NETWORK
TITLE =R5_Kreislauf_ohne_aussen  Rinser CIP-Kreis ohne pulsierenden
// Act 006
// Box           : Rinser5
// Output address: Q172.3
      CALL FC    70 (
           UnitNo                   := #UnitNo,
           ActRec                   := DB2650.R5_Kreislauf_ohne_aussen,
           Typ                      := 0,
           FBa                      := #xTmp,
           FBa2                     := #xTmp,
           Out                      := Q    172.3);

NETWORK
TITLE =R5_Kreislauf_mit_aussen  Rinser CIP-Kreis mit pulsierenden
// Act 007
// Box           : Rinser5
// Output address: Q172.4
      CALL FC    70 (
           UnitNo                   := #UnitNo,
           ActRec                   := DB2650.R5_Kreislauf_mit_aussen,
           Typ                      := 0,
           FBa                      := #xTmp,
           FBa2                     := #xTmp,
           Out                      := Q    172.4);

NETWORK
TITLE =R5_Grundstellung  Rinser A5 Maschine Grundstellung (Impuls)
// Act 008
// Box           : Rinser5
// Output address: Q172.2
      CALL FC    70 (
           UnitNo                   := #UnitNo,
           ActRec                   := DB2650.R5_Grundstellung,
           Typ                      := 0,
           FBa                      := #xTmp,
           FBa2                     := #xTmp,
           Out                      := Q    172.2);

NETWORK
TITLE =R5_Drainagestellung  Rinser A5 Drainagestellung (Impuls)
// Act 009
// Box           : Rinser5
// Output address: Q172.5
      CALL FC    70 (
           UnitNo                   := #UnitNo,
           ActRec                   := DB2650.R5_Drainagestellung,
           Typ                      := 0,
           FBa                      := #xTmp,
           FBa2                     := #xTmp,
           Out                      := Q    172.5);

NETWORK
TITLE =F5_Kreislauf_o_puls  Füller CIP-Kreis ohne pulsierenden Ablauf
// Act 010
// Box           : Füller5
// Output address: Q196.2
      CALL FC    70 (
           UnitNo                   := #UnitNo,
           ActRec                   := DB2650.F5_Kreislauf_o_puls,
           Typ                      := 0,
           FBa                      := #xTmp,
           FBa2                     := #xTmp,
           Out                      := Q    196.2);

NETWORK
TITLE =F5_Kreislauf_m_puls  Füller CIP-Kreis mit pulsierenden Ablauf
// Act 011
// Box           : Füller5
// Output address: Q196.3
      CALL FC    70 (
           UnitNo                   := #UnitNo,
           ActRec                   := DB2650.F5_Kreislauf_m_puls,
           Typ                      := 0,
           FBa                      := #xTmp,
           FBa2                     := #xTmp,
           Out                      := Q    196.3);

NETWORK
TITLE =F5_Randvollstellung  Füller A5 Randvollstellung Standdesinfektio
// Act 012
// Box           : Füller5
// Output address: Q196.4
      CALL FC    70 (
           UnitNo                   := #UnitNo,
           ActRec                   := DB2650.F5_Randvollstellung,
           Typ                      := 0,
           FBa                      := #xTmp,
           FBa2                     := #xTmp,
           Out                      := Q    196.4);

NETWORK
TITLE =F5_Klarspuelen_o_CIP_Beh  Füller A5 Klarspülen ohne CIP-Behälter
// Act 013
// Box           : Füller5
// Output address: Q196.5
      CALL FC    70 (
           UnitNo                   := #UnitNo,
           ActRec                   := DB2650.F5_Klarspuelen_o_CIP_Beh,
           Typ                      := 0,
           FBa                      := #xTmp,
           FBa2                     := #xTmp,
           Out                      := Q    196.5);

NETWORK
TITLE =F5_Ausschub_m_Sterilluft  Füller Ausschubprogramm mit Sterilluft
// Act 014
// Box           : Füller5
// Output address: Q196.6
      CALL FC    70 (
           UnitNo                   := #UnitNo,
           ActRec                   := DB2650.F5_Ausschub_m_Sterilluft,
           Typ                      := 0,
           FBa                      := #xTmp,
           FBa2                     := #xTmp,
           Out                      := Q    196.6);

NETWORK
TITLE =F5_Ausschub_m_CO2  Füller A5 Ausschubprogramm mit CO2
// Act 015
// Box           : Füller5
// Output address: Q196.7
      CALL FC    70 (
           UnitNo                   := #UnitNo,
           ActRec                   := DB2650.F5_Ausschub_m_CO2,
           Typ                      := 0,
           FBa                      := #xTmp,
           FBa2                     := #xTmp,
           Out                      := Q    196.7);

NETWORK
TITLE =F5_Grundstellung  Füller A5 Maschine Grundstellung (Impuls)
// Act 016
// Box           : Füller5
// Output address: Q197.0
      CALL FC    70 (
           UnitNo                   := #UnitNo,
           ActRec                   := DB2650.F5_Grundstellung,
           Typ                      := 0,
           FBa                      := #xTmp,
           FBa2                     := #xTmp,
           Out                      := Q    197.0);

NETWORK
TITLE =F5_Drainagestellung  Füller A5 Drainagestellung (Impuls)
// Act 017
// Box           : Füller5
// Output address: Q197.1
      CALL FC    70 (
           UnitNo                   := #UnitNo,
           ActRec                   := DB2650.F5_Drainagestellung,
           Typ                      := 0,
           FBa                      := #xTmp,
           FBa2                     := #xTmp,
           Out                      := Q    197.1);

NETWORK
TITLE =F5_Bypass  Füller A5 Bypass (Impuls)
// Act 018
// Box           : Füller5
// Output address: Q197.2
      CALL FC    70 (
           UnitNo                   := #UnitNo,
           ActRec                   := DB2650.F5_Bypass,
           Typ                      := 0,
           FBa                      := #xTmp,
           FBa2                     := #xTmp,
           Out                      := Q    197.2);

NETWORK
TITLE =A5_RR1  Reinigungsrücklauf Anlage 5 zu Kreis 1
// Act 020
// Box           : VSRR1-3
// Input address : I84.0
// Output address: Q84.0
      CALL FC    70 (
           UnitNo                   := #UnitNo,
           ActRec                   := DB2650.A5_RR1,
           Typ                      := 1,
           FBa                      := #xTmp,
           FBa2                     := I     84.0,
           Out                      := Q     84.0);

NETWORK
TITLE =A5_RR2  Reinigungsrücklauf Anlage 5 zu Kreis 2
// Act 021
// Box           : VSRR1-3
// Input address : I84.1
// Output address: Q84.1
      CALL FC    70 (
           UnitNo                   := #UnitNo,
           ActRec                   := DB2650.A5_RR2,
           Typ                      := 1,
           FBa                      := #xTmp,
           FBa2                     := I     84.1,
           Out                      := Q     84.1);

NETWORK
TITLE =A5_RR3  Reinigungsrücklauf Anlage 5 zu Kreis 3
// Act 022
// Box           : VSRR1-3
// Input address : I84.2
// Output address: Q84.2
      CALL FC    70 (
           UnitNo                   := #UnitNo,
           ActRec                   := DB2650.A5_RR3,
           Typ                      := 1,
           FBa                      := #xTmp,
           FBa2                     := I     84.2,
           Out                      := Q     84.2);

NETWORK
TITLE =M5_Grundstellung  Mixer A5 Grundstellung (Impuls)
// Act 023
// Box           : Mixer5
// Output address: Q198.0
      CALL FC    70 (
           UnitNo                   := #UnitNo,
           ActRec                   := DB2650.M5_Grundstellung,
           Typ                      := 0,
           FBa                      := #xTmp,
           FBa2                     := #xTmp,
           Out                      := Q    198.0);

NETWORK
TITLE =M5_Drainagestellung  Mixer A5 Drainagestellung (Impuls)
// Act 024
// Box           : Mixer5
// Output address: Q198.1
      CALL FC    70 (
           UnitNo                   := #UnitNo,
           ActRec                   := DB2650.M5_Drainagestellung,
           Typ                      := 0,
           FBa                      := #xTmp,
           FBa2                     := #xTmp,
           Out                      := Q    198.1);

NETWORK
TITLE =M5_Ausspritzen_o_Ablauf  MixerAusspritzen ohne Ablauf
// Act 025
// Box           : Mixer5
// Output address: Q198.2
      CALL FC    70 (
           UnitNo                   := #UnitNo,
           ActRec                   := DB2650.M5_Ausspritzen_o_Ablauf,
           Typ                      := 0,
           FBa                      := #xTmp,
           FBa2                     := #xTmp,
           Out                      := Q    198.2);

NETWORK
TITLE =M5_Ausspritzen_m_Ablauf  Mixer A5 Ausspritzen mit Ablauf (Impuls
// Act 026
// Box           : Mixer5
// Output address: Q198.3
      CALL FC    70 (
           UnitNo                   := #UnitNo,
           ActRec                   := DB2650.M5_Ausspritzen_m_Ablauf,
           Typ                      := 0,
           FBa                      := #xTmp,
           FBa2                     := #xTmp,
           Out                      := Q    198.3);

NETWORK
TITLE =M5_Fluten_o_Ablauf  Mixer A5 Fluten ohne Ablauf (Impuls)
// Act 027
// Box           : Mixer5
// Output address: Q198.4
      CALL FC    70 (
           UnitNo                   := #UnitNo,
           ActRec                   := DB2650.M5_Fluten_o_Ablauf,
           Typ                      := 0,
           FBa                      := #xTmp,
           FBa2                     := #xTmp,
           Out                      := Q    198.4);

NETWORK
TITLE =M5_Fluten_m_Ablauf  Mixer A5 Fluten mit Ablauf (Impuls)
// Act 028
// Box           : Mixer5
// Output address: Q198.5
      CALL FC    70 (
           UnitNo                   := #UnitNo,
           ActRec                   := DB2650.M5_Fluten_m_Ablauf,
           Typ                      := 0,
           FBa                      := #xTmp,
           FBa2                     := #xTmp,
           Out                      := Q    198.5);

NETWORK
TITLE =M5_Randvollstellung  Mixer A5 Randvollstellung (Impuls)
// Act 029
// Box           : Mixer5
// Output address: Q198.6
      CALL FC    70 (
           UnitNo                   := #UnitNo,
           ActRec                   := DB2650.M5_Randvollstellung,
           Typ                      := 0,
           FBa                      := #xTmp,
           FBa2                     := #xTmp,
           Out                      := Q    198.6);

NETWORK
TITLE =M5_Abpumpen  Mixer A5 Abpumpen (Impuls)
// Act 030
// Box           : Mixer5
// Output address: Q198.7
      CALL FC    70 (
           UnitNo                   := #UnitNo,
           ActRec                   := DB2650.M5_Abpumpen,
           Typ                      := 0,
           FBa                      := #xTmp,
           FBa2                     := #xTmp,
           Out                      := Q    198.7);

NETWORK
TITLE =M5_Klarspuelen  Mixer A5 Klarspülen
// Act 031
// Box           : Mixer5
// Output address: Q199.0
      CALL FC    70 (
           UnitNo                   := #UnitNo,
           ActRec                   := DB2650.M5_Klarspuelen,
           Typ                      := 0,
           FBa                      := #xTmp,
           FBa2                     := #xTmp,
           Out                      := Q    199.0);

END_FUNCTION_BLOCK

FUNCTION_BLOCK FB 1651
TITLE =U065: Packaging Plant 5
FAMILY : BOTEC_F1
NAME : UniE
VERSION : 1.2


VAR_TEMP
  CIP : BOOL ;	//CIP active
  UNIM : BOOL ;	//Unit Not In Maintenance
  GenRel : BOOL ;	//general OK (emergency and maintenance OK)
  EStopOK : BOOL ;	//emergency OK
  UnitNo : INT ;	//unit number
  xTmp : BOOL ;	//Temporary Bool
  iTmp : INT ;	//Temporary INT
  rTmp : REAL ;	//Temporary REAL
  dTmp : DINT ;	//Temporary DINT (free for general use)
  RetValInt : INT ;	//return value
END_VAR
BEGIN
NETWORK
TITLE =General

      SET   ;
// Simulation ---------------------------------------------------------------
      A     DB1651.DBX 1357.7;
      CC    FB  1659; // "U065Sim"
      A     DB1651.DBX   17.3;
      =     DB1651.DBX 1357.7; //Help bit for simulation

// get unit number ----------------------------------------------------------
      L     DB1650.DBW    0;
      T     #UnitNo;

// CIP ----------------------------------------------------------------------
      L     DB1651.DBD   54;
      L     0;
      <D    ;
      =     #CIP;

// emergency OK -------------------------------------------------------------
      A     DB1655.DBX   27.0; //Emergency Stop OK
      =     #EStopOK;

// Write Unit in Maintenance ------------------------------------------------

      AN    DB1651.DBX   69.7;
      =     #UNIM;

// emergency and maintenance OK ---------------------------------------------
      A     #EStopOK;
      A     #UNIM;
      =     #GenRel;

// communication ------------------------------------------------------------
      UC    FB  1655; // U065Com

NETWORK
TITLE =Analog Inputs

      NOP   0;

// ----------------------------------------------------------
// A5_TI1
// ----------------------------------------------------------
//      L     ID   352
//      T     "U065AnID".A5_TI1.ValRaw
      SET   ;
      R     DB2653.DBX  143.5;

      L     DB1651.DBD 1118; // !!! insert correct SFM !!!
      T     DB2653.DBD  238;

      SET   ;
      =     DB2653.DBX  141.5;


NETWORK
TITLE =Universal Value

      NOP   0;

// ----------------------------------------------------------
// unv001 Process Status
// ----------------------------------------------------------
// process value to UnV
//      L     0.000000e+000
//      T     "U065UnVD".unv001.ValExt

// ----------------------------------------------------------
// unv002 Universal Value 02
// ----------------------------------------------------------
// process value to UnV
//      L     0.000000e+000
//      T     "U065UnVD".unv002.ValExt

// ----------------------------------------------------------
// unv003 Universal Value 03
// ----------------------------------------------------------
// process value to UnV
//      L     0.000000e+000
//      T     "U065UnVD".unv003.ValExt

// ----------------------------------------------------------
// unv004 Universal Value 04
// ----------------------------------------------------------
// process value to UnV
//      L     0.000000e+000
//      T     "U065UnVD".unv004.ValExt

NETWORK
TITLE =Special Input

      NOP   0;

// ----------------------------------------------------------
// A5_MIXER_CIP_BEREIT Koppelsignal von Mixer 5 CIP-Bereitschaft (Dauersignal)
// ----------------------------------------------------------
      A     DB2650.DBX  102.6;
      =     DB2651.DBX   81.4;
      SET   ;
      =     DB2651.DBX   81.5;


// ----------------------------------------------------------
// A5_MIXER_VOLL Koppelsignal von Mixer 5 Mixer voll
// ----------------------------------------------------------
//      CLR
//      =     "U065SpID".A5_MIXER_VOLL.EAl
//      =     "U065SpID".A5_MIXER_VOLL.Pre

// ----------------------------------------------------------
// A5_MIXER_LEER Koppelsignal von Mixer 5 Mixer leer
// ----------------------------------------------------------
//      CLR
//      =     "U065SpID".A5_MIXER_LEER.EAl
//      =     "U065SpID".A5_MIXER_LEER.Pre

// ----------------------------------------------------------
// A5_MIXER_Anforderung Koppelsignal von Mixer 5 Anforderung Nachsp.
// ----------------------------------------------------------
//      CLR
//      =     "U065SpID".A5_MIXER_Anforderung.EAl
//      =     "U065SpID".A5_MIXER_Anforderung.Pre

// ----------------------------------------------------------
// M5_WATCHDOG Koppelsignal von Mixer 5 WATCHDOG
// ----------------------------------------------------------
//      CLR
//      =     "U065SpID".M5_WATCHDOG.EAl
//      =     "U065SpID".M5_WATCHDOG.Pre

// ----------------------------------------------------------
// A5_SS_FRG_MOLCH Anlage 5 Schlüsselschalter Freigabe Molch
// ----------------------------------------------------------
//      CLR
//      =     "U065SpID".A5_SS_FRG_MOLCH.EAl
//      =     "U065SpID".A5_SS_FRG_MOLCH.Pre

// ----------------------------------------------------------
// E195_7 Anlage 5 Reserve 7 Ende Ventilschrank A5
// ----------------------------------------------------------
//      CLR
//      =     "U065SpID".E195_7.EAl
//      =     "U065SpID".E195_7.Pre

// ----------------------------------------------------------
// A5_LDT_PROD
// ----------------------------------------------------------
//      CLR
//      =     "U065SpID".A5_LDT_PROD.EAl
//      =     "U065SpID".A5_LDT_PROD.Pre

// ----------------------------------------------------------
// A5_LDT_QUITT_CIP
// ----------------------------------------------------------
//      CLR
//      =     "U065SpID".A5_LDT_QUITT_CIP.EAl
//      =     "U065SpID".A5_LDT_QUITT_CIP.Pre

// ----------------------------------------------------------
// A5_DT_START
// ----------------------------------------------------------
//      CLR
//      =     "U065SpID".A5_DT_START.EAl
//      =     "U065SpID".A5_DT_START.Pre

// ----------------------------------------------------------
// A5_FUELLER_LAEUFT Koppelsignal von Füller 5 Füller läuft (Dauersignal)
// ----------------------------------------------------------
//      CLR
//      =     "U065SpID".A5_FUELLER_LAEUFT.EAl
//      =     "U065SpID".A5_FUELLER_LAEUFT.Pre

// ----------------------------------------------------------
// A5_FUELLER_LEER Koppelsignal von Füller 5 Füller leer (Impuls)
// ----------------------------------------------------------
//      CLR
//      =     "U065SpID".A5_FUELLER_LEER.EAl
//      =     "U065SpID".A5_FUELLER_LEER.Pre

// ----------------------------------------------------------
// A5_FUELLER_VOLL Koppelsignal von Füller 5 Füller voll (Impuls)
// ----------------------------------------------------------
//      CLR
//      =     "U065SpID".A5_FUELLER_VOLL.EAl
//      =     "U065SpID".A5_FUELLER_VOLL.Pre

// ----------------------------------------------------------
// A5_FUELLER_KLARSPUELEN Koppelsignal von Füller 5 Klarspülen
// ----------------------------------------------------------
//      CLR
//      =     "U065SpID".A5_FUELLER_KLARSPUELEN.EAl
//      =     "U065SpID".A5_FUELLER_KLARSPUELEN.Pre

// ----------------------------------------------------------
// F5_WATCHDOG Koppelsignal von Füller 5 WATCHDOG
// ----------------------------------------------------------
//      CLR
//     =     "U065SpID".F5_WATCHDOG.EAl
//     =     "U065SpID".F5_WATCHDOG.Pre

// ----------------------------------------------------------
// A5_RINSER_LAEUFT Koppelsignal von Rinser 5 Rinser läuft (Dauersignal)
// ----------------------------------------------------------
//      CLR
//      =     "U065SpID".A5_RINSER_LAEUFT.EAl
//      =     "U065SpID".A5_RINSER_LAEUFT.Pre

// ----------------------------------------------------------
// R5_WATCHDOG Koppelsignal von Rinser 5 WATCHDOG
// ----------------------------------------------------------
//      CLR
//      =     "U065SpID".R5_WATCHDOG.EAl
//      =     "U065SpID".R5_WATCHDOG.Pre

NETWORK
TITLE =Messages

      NOP   0;

// ----------------------------------------------------------
// msg001 Message 01
// ----------------------------------------------------------
      SET   ;
      R     DB2657.DBX   80.7;
      =     DB2657.DBX   81.4;

      CLR   ;
      =     DB2657.DBX   82.7;

// ----------------------------------------------------------
// msg002 Message 02
// ----------------------------------------------------------
      SET   ;
      R     DB2657.DBX  140.7;
      =     DB2657.DBX  141.4;

      CLR   ;
      =     DB2657.DBX  142.7;

// ----------------------------------------------------------
// msg003 Message 03
// ----------------------------------------------------------
      SET   ;
      R     DB2657.DBX  200.7;
      =     DB2657.DBX  201.4;

      CLR   ;
      =     DB2657.DBX  202.7;

NETWORK
TITLE =Sequence organisation

      CLR   ;
      =     M    122.2;

// SFM supply ----------------------------------------------------------------

// analog value to SFM spare -----------------------
      L     DB2653.DBD  146;
      T     DB1651.DBD 1122; // !!! insert correct SFM !!!

// sequencer ----------------------------------------------------------------
      A     DB1653.DBX   43.1;
      S     DB1653.DBX   97.3;

      CALL FC    40 (
           UnitNo                   := #UnitNo);

NETWORK
TITLE =Auto / Manual

      SET   ;
      AN    M    122.2;
      JC    MODE;
      AN    M    120.1;

// assign actuator mode
      AN    M    120.1;
      =     DB2650.DBX  105.4;
      =     DB2650.DBX  185.4;
      S     DB2650.DBX  265.4;
      =     DB2650.DBX  345.4;
      S     DB2650.DBX  425.4;
      =     DB2650.DBX  505.4;
      =     DB2650.DBX  585.4;
      =     DB2650.DBX  665.4;
      =     DB2650.DBX  745.4;
      =     DB2650.DBX  825.4;
      =     DB2650.DBX  905.4;
      =     DB2650.DBX  985.4;
      =     DB2650.DBX 1065.4;
      =     DB2650.DBX 1145.4;
      =     DB2650.DBX 1225.4;
      =     DB2650.DBX 1305.4;
      =     DB2650.DBX 1385.4;
      =     DB2650.DBX 1465.4;
      =     DB2650.DBX 1545.4;
      =     DB2650.DBX 1625.4;
      =     DB2650.DBX 1705.4;
      =     DB2650.DBX 1785.4;
      =     DB2650.DBX 1865.4;
      =     DB2650.DBX 1945.4;
      =     DB2650.DBX 2025.4;
      =     DB2650.DBX 2105.4;
      =     DB2650.DBX 2185.4;
      =     DB2650.DBX 2265.4;
      =     DB2650.DBX 2345.4;
      =     DB2650.DBX 2425.4;
      =     DB2650.DBX 2505.4;




MODE: SET   ;

NETWORK
TITLE =A5_RP1 Rücklaufpumpe Anlage 5
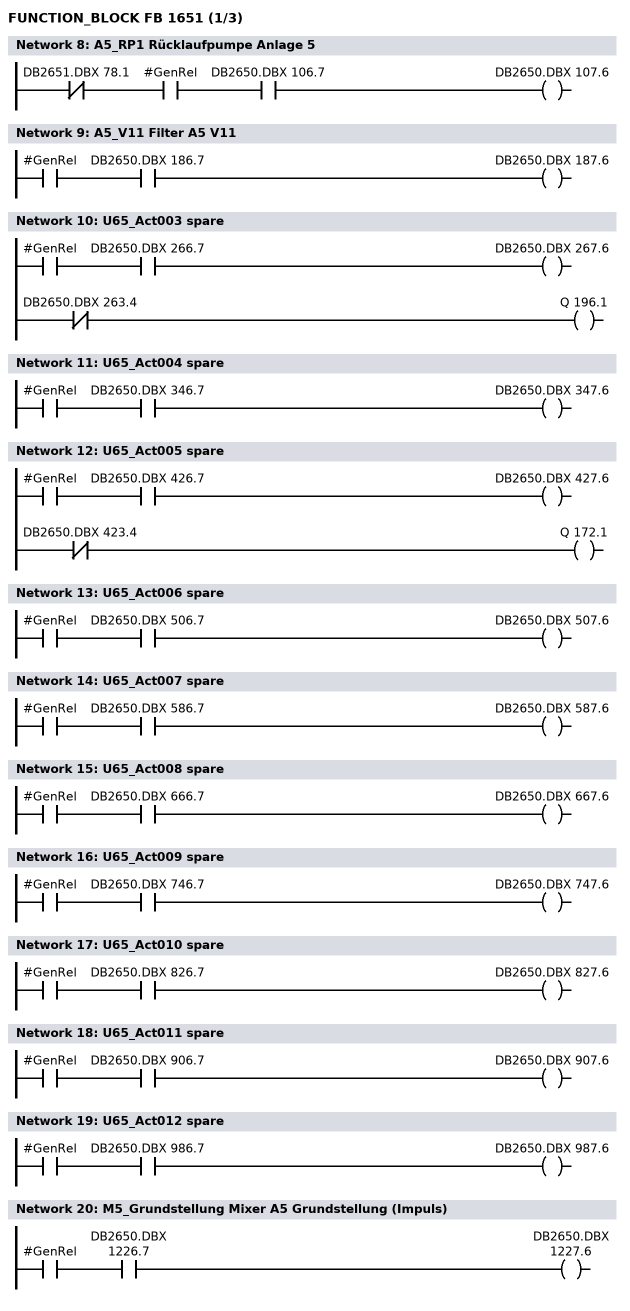

//      A     "U065SpID".A5_FS1.Sig
      AN    DB2651.DBX   78.1;

      A     #GenRel;
      A     DB2650.DBX  106.7;
      =     DB2650.DBX  107.6;
NETWORK
TITLE =A5_V11 Filter A5 V11

      A     #GenRel;
      A     DB2650.DBX  186.7;
      =     DB2650.DBX  187.6;
NETWORK
TITLE =U65_Act003 spare

      A     #GenRel;
      A     DB2650.DBX  266.7;
      =     DB2650.DBX  267.6;

      AN    DB2650.DBX  263.4;
      =     Q    196.1;
NETWORK
TITLE =U65_Act004 spare

      A     #GenRel;
      A     DB2650.DBX  346.7;
      =     DB2650.DBX  347.6;
NETWORK
TITLE =U65_Act005 spare

      A     #GenRel;
      A     DB2650.DBX  426.7;
      =     DB2650.DBX  427.6;

      AN    DB2650.DBX  423.4;
      =     Q    172.1;
NETWORK
TITLE =U65_Act006 spare

      A     #GenRel;
      A     DB2650.DBX  506.7;
      =     DB2650.DBX  507.6;
NETWORK
TITLE =U65_Act007 spare

      A     #GenRel;
      A     DB2650.DBX  586.7;
      =     DB2650.DBX  587.6;
NETWORK
TITLE =U65_Act008 spare

      A     #GenRel;
      A     DB2650.DBX  666.7;
      =     DB2650.DBX  667.6;
NETWORK
TITLE =U65_Act009 spare

      A     #GenRel;
      A     DB2650.DBX  746.7;
      =     DB2650.DBX  747.6;
NETWORK
TITLE =U65_Act010 spare

      A     #GenRel;
      A     DB2650.DBX  826.7;
      =     DB2650.DBX  827.6;
NETWORK
TITLE =U65_Act011 spare

      A     #GenRel;
      A     DB2650.DBX  906.7;
      =     DB2650.DBX  907.6;
NETWORK
TITLE =U65_Act012 spare

      A     #GenRel;
      A     DB2650.DBX  986.7;
      =     DB2650.DBX  987.6;
NETWORK
TITLE =M5_Grundstellung Mixer A5 Grundstellung (Impuls)

      A     #GenRel;
      A     DB2650.DBX 1226.7;
      =     DB2650.DBX 1227.6;
NETWORK
TITLE =M5_Drainagestellung Mixer A5 Drainagestellung (Impuls)
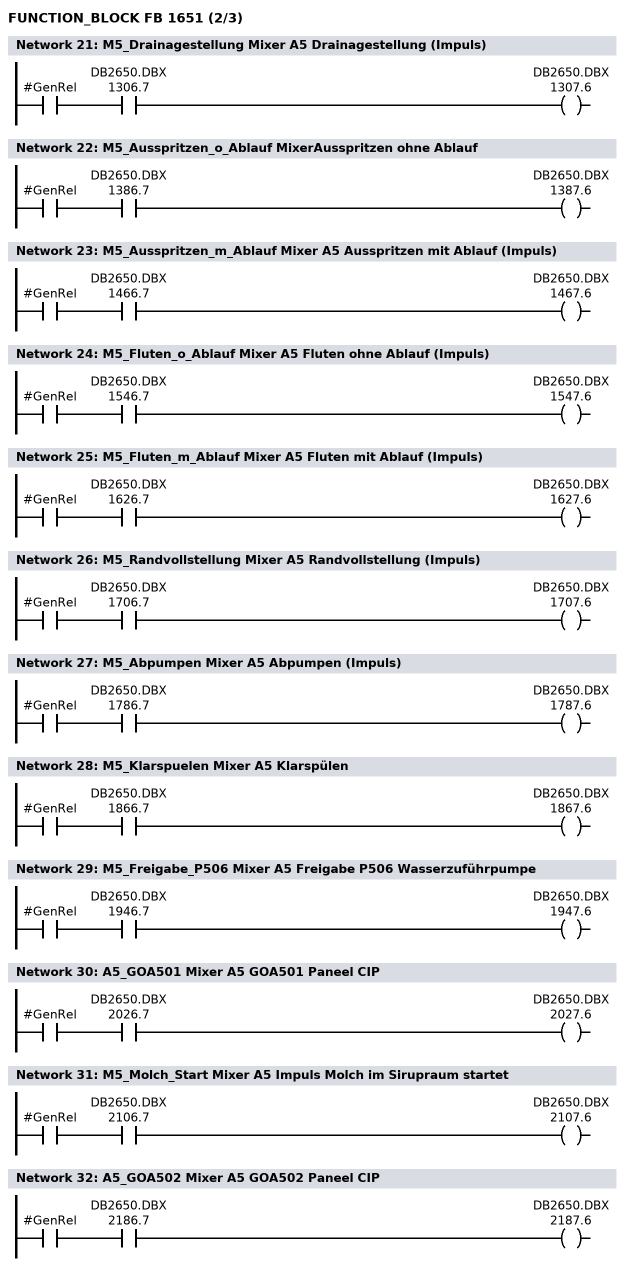

      A     #GenRel;
      A     DB2650.DBX 1306.7;
      =     DB2650.DBX 1307.6;
NETWORK
TITLE =M5_Ausspritzen_o_Ablauf MixerAusspritzen ohne Ablauf

      A     #GenRel;
      A     DB2650.DBX 1386.7;
      =     DB2650.DBX 1387.6;
NETWORK
TITLE =M5_Ausspritzen_m_Ablauf Mixer A5 Ausspritzen mit Ablauf (Impuls)

      A     #GenRel;
      A     DB2650.DBX 1466.7;
      =     DB2650.DBX 1467.6;
NETWORK
TITLE =M5_Fluten_o_Ablauf Mixer A5 Fluten ohne Ablauf (Impuls)

      A     #GenRel;
      A     DB2650.DBX 1546.7;
      =     DB2650.DBX 1547.6;
NETWORK
TITLE =M5_Fluten_m_Ablauf Mixer A5 Fluten mit Ablauf (Impuls)

      A     #GenRel;
      A     DB2650.DBX 1626.7;
      =     DB2650.DBX 1627.6;
NETWORK
TITLE =M5_Randvollstellung Mixer A5 Randvollstellung (Impuls)

      A     #GenRel;
      A     DB2650.DBX 1706.7;
      =     DB2650.DBX 1707.6;
NETWORK
TITLE =M5_Abpumpen Mixer A5 Abpumpen (Impuls)

      A     #GenRel;
      A     DB2650.DBX 1786.7;
      =     DB2650.DBX 1787.6;
NETWORK
TITLE =M5_Klarspuelen Mixer A5 Klarspülen

      A     #GenRel;
      A     DB2650.DBX 1866.7;
      =     DB2650.DBX 1867.6;
NETWORK
TITLE =M5_Freigabe_P506 Mixer A5 Freigabe P506 Wasserzuführpumpe

      A     #GenRel;
      A     DB2650.DBX 1946.7;
      =     DB2650.DBX 1947.6;
NETWORK
TITLE =A5_GOA501 Mixer A5 GOA501 Paneel CIP

      A     #GenRel;
      A     DB2650.DBX 2026.7;
      =     DB2650.DBX 2027.6;
NETWORK
TITLE =M5_Molch_Start Mixer A5 Impuls Molch im Sirupraum startet

      A     #GenRel;
      A     DB2650.DBX 2106.7;
      =     DB2650.DBX 2107.6;
NETWORK
TITLE =A5_GOA502 Mixer A5 GOA502 Paneel CIP

      A     #GenRel;
      A     DB2650.DBX 2186.7;
      =     DB2650.DBX 2187.6;
NETWORK
TITLE =A5_GOA503 Mixer A5 GOA503 Paneel CIP
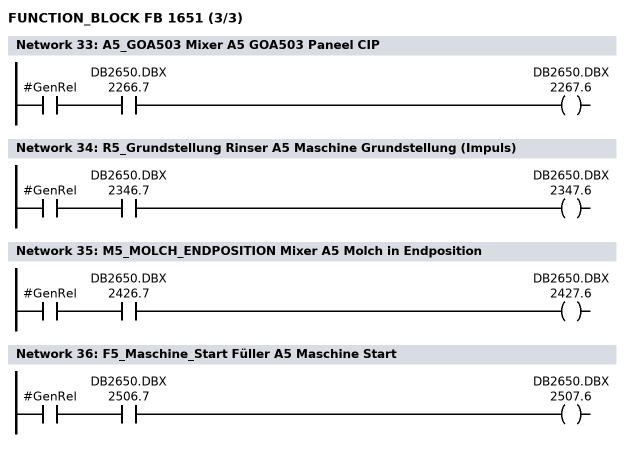

      A     #GenRel;
      A     DB2650.DBX 2266.7;
      =     DB2650.DBX 2267.6;
NETWORK
TITLE =R5_Grundstellung Rinser A5 Maschine Grundstellung (Impuls)

      A     #GenRel;
      A     DB2650.DBX 2346.7;
      =     DB2650.DBX 2347.6;
NETWORK
TITLE =M5_MOLCH_ENDPOSITION Mixer A5 Molch in Endposition

      A     #GenRel;
      A     DB2650.DBX 2426.7;
      =     DB2650.DBX 2427.6;
NETWORK
TITLE =F5_Maschine_Start Füller A5 Maschine Start

      A     #GenRel;
      A     DB2650.DBX 2506.7;
      =     DB2650.DBX 2507.6;
END_FUNCTION_BLOCK

FUNCTION_BLOCK FB 1670
TITLE =U067: Abfüllanlage  7
FAMILY : BOTEC_F1
NAME : U067A
VERSION : 2.1


VAR_TEMP
  EStopOK : BOOL ;	//auxiliary flag
  CIP : BOOL ;	//CIP Program Selected
  xTmp : BOOL ;	//Temporary Bool(free for general use)
  DummyBool : BOOL ;	//Temporary Bool(free for general use)
  UnitNo : INT ;	//unit number
  UnitFB : INT ;	//unit expansion FB number
  rTmp : REAL ;	//Temporary REAL (free for general use)
  iTmp : INT ;	//Temporary INT (free for general use)
  DummyInt : INT ;	//Temporary INT (free for general use)
  dTmp : DINT ;	//Temporary DINT (free for general use)
END_VAR
BEGIN
NETWORK
TITLE =general

      CLR   ;
      =     #xTmp;
      =     #EStopOK;

      L     DB1670.DBW    0;
      T     #UnitNo;
      L     DB1670.DBW    2;
      T     #UnitFB;

NETWORK
TITLE =Universal value

      NOP   0;
// unv001 UnV 001 Process Status
      CALL FC    27 (
           UnitNo                   := #UnitNo,
           UnVRec                   := DB2675.unv001,
           ValExt                   := DB2675.DBD  234);

// unv002 UnV 002 Universal Value 02
      CALL FC    27 (
           UnitNo                   := #UnitNo,
           UnVRec                   := DB2675.unv002,
           ValExt                   := DB2675.DBD  362);

// unv003 UnV 003 Universal Value 03
      CALL FC    27 (
           UnitNo                   := #UnitNo,
           UnVRec                   := DB2675.unv003,
           ValExt                   := DB2675.DBD  490);

// unv004 UnV 004 Universal Value 04
      CALL FC    27 (
           UnitNo                   := #UnitNo,
           UnVRec                   := DB2675.unv004,
           ValExt                   := DB2675.DBD  618);

NETWORK
TITLE =special inputs

      NOP   0;
// FS_A7FS1 SpI 001 STROEMUNGSSCHALTER A7
      CALL FC    14 (
           UnitNo                   := #UnitNo,
           SpIRec                   := DB2671.FS_A7FS1,
           SpIBit                   := I     27.0);

// A7_FUELLER_LAEUFT SpI 002 Fueller 7 laeuft
      CALL FC    14 (
           UnitNo                   := #UnitNo,
           SpIRec                   := DB2671.A7_FUELLER_LAEUFT,
           SpIBit                   := I     76.1);

// A7_MIXER_CIP_BEREIT SpI 003 Mixer Anlage 7 CIP-Bereit
      CALL FC    14 (
           UnitNo                   := #UnitNo,
           SpIRec                   := DB2671.A7_MIXER_CIP_BEREIT,
           SpIBit                   := I     78.0);

// A7_MIXER_VOLL SpI 004 Mixer Anlage 7 voll
      CALL FC    14 (
           UnitNo                   := #UnitNo,
           SpIRec                   := DB2671.A7_MIXER_VOLL,
           SpIBit                   := I     78.2);

// A7_MIXER_LEER SpI 005 Mixer Anlage 7 leer
      CALL FC    14 (
           UnitNo                   := #UnitNo,
           SpIRec                   := DB2671.A7_MIXER_LEER,
           SpIBit                   := I     78.1);

// A7_MIXER_ANF_SIRUP SpI 006 Mixer Anlage 7 Anforderung Sirup
      CALL FC    14 (
           UnitNo                   := #UnitNo,
           SpIRec                   := DB2671.A7_MIXER_ANF_SIRUP,
           SpIBit                   := I     78.3);

// A7_FUELLER_CIP_BEREIT SpI 007 Fueller 7 CIP-Bereit
      CALL FC    14 (
           UnitNo                   := #UnitNo,
           SpIRec                   := DB2671.A7_FUELLER_CIP_BEREIT,
           SpIBit                   := I     76.0);

// A7_SS_FRG_MOLCH SpI 009 Anlage 7 Schlüsselschalter Freigabe Molch
      CALL FC    14 (
           UnitNo                   := #UnitNo,
           SpIRec                   := DB2671.A7_SS_FRG_MOLCH,
           SpIBit                   := I     27.4);

// A7_FUELLER_LEER SpI 011 Fueller 7 leer (Impuls)
      CALL FC    14 (
           UnitNo                   := #UnitNo,
           SpIRec                   := DB2671.A7_FUELLER_LEER,
           SpIBit                   := I     76.2);

// GOA_703 SpI 012 Meldung an Fueller/Mixer Anl.7
      CALL FC    14 (
           UnitNo                   := #UnitNo,
           SpIRec                   := DB2671.A7_FUELLER_VOLL,
           SpIBit                   := I     76.3);//"GOA_703"

// A7_RINSER_CIP_BEREIT SpI 013 Rinser Anlage 7 CIP-Bereit
      CALL FC    14 (
           UnitNo                   := #UnitNo,
           SpIRec                   := DB2671.A7_RINSER_CIP_BEREIT,
           SpIBit                   := I     77.0);

// A7_RINSER_LAEUFT SpI 014 Rinser Anlage 7 laeuft
      CALL FC    14 (
           UnitNo                   := #UnitNo,
           SpIRec                   := DB2671.A7_RINSER_LAEUFT,
           SpIBit                   := I     77.1);

// EA7_K1_Handklappe SpI 015 Handklappe Fueller 7
      CALL FC    14 (
           UnitNo                   := #UnitNo,
           SpIRec                   := DB2671.EA7_K1_Handklappe,
           SpIBit                   := I     27.1);

NETWORK
TITLE =messages

      NOP   0;
// msg001 Msg 001 Message 01
      CALL FC    16 (
           UnitNo                   := #UnitNo,
           MsgRec                   := DB2677.msg001,
           MsgBit                   := DB2677.DBX   82.7);

// msg002 Msg 002 Message 02
      CALL FC    16 (
           UnitNo                   := #UnitNo,
           MsgRec                   := DB2677.msg002,
           MsgBit                   := DB2677.DBX  142.7);

// msg003 Msg 003 Message 03
      CALL FC    16 (
           UnitNo                   := #UnitNo,
           MsgRec                   := DB2677.msg003,
           MsgBit                   := DB2677.DBX  202.7);

NETWORK
TITLE =unit supply

      UC    FB [#UnitFB];

NETWORK
TITLE =A7_RRP1  CIP Rücklaufpumpe Anlage 7
// Act 001
// Box           : VSA7
// Input address : I25.7
// Output address: Q47.7
      CALL FC    70 (
           UnitNo                   := #UnitNo,
           ActRec                   := DB2670.A7_RRP1,
           Typ                      := 1,
           FBa                      := #xTmp,
           FBa2                     := I     25.7,
           Out                      := Q     47.7);

NETWORK
TITLE =F7_Maschine_Start  Fueller 7 Start
// Act 002
// Box           : FRM-A7
// Output address: Q54.0
      CALL FC    70 (
           UnitNo                   := #UnitNo,
           ActRec                   := DB2670.F7_Maschine_Start,
           Typ                      := 0,
           FBa                      := #xTmp,
           FBa2                     := #xTmp,
           Out                      := Q     54.0);

NETWORK
TITLE =F7_Maschine_Stop  Fueller 7 Stop
// Act 003
// Box           : FRM-A7
// Output address: Q54.1
      CALL FC    70 (
           UnitNo                   := #UnitNo,
           ActRec                   := DB2670.F7_Maschine_Stop,
           Typ                      := 0,
           FBa                      := #xTmp,
           FBa2                     := #xTmp,
           Out                      := #xTmp);

NETWORK
TITLE =R7_START_IMPULS  Rinser 7 Start
// Act 004
// Box           : FRM-A7
// Output address: Q56.0
      CALL FC    70 (
           UnitNo                   := #UnitNo,
           ActRec                   := DB2670.R7_START_IMPULS,
           Typ                      := 0,
           FBa                      := #xTmp,
           FBa2                     := #xTmp,
           Out                      := Q     56.0);

NETWORK
TITLE =R7_STOP  Rinser 7 Stop
// Act 005
// Box           : FRM-A7
// Output address: Q56.1
      CALL FC    70 (
           UnitNo                   := #UnitNo,
           ActRec                   := DB2670.R7_STOP,
           Typ                      := 0,
           FBa                      := #xTmp,
           FBa2                     := #xTmp,
           Out                      := #xTmp);

NETWORK
TITLE =R7_Kreislauf_ohne_aussen  Prog.schritt 15 CIP Krsl.o.ausse.
// Act 006
// Box           : FRM-A7
// Output address: Q56.3
      CALL FC    70 (
           UnitNo                   := #UnitNo,
           ActRec                   := DB2670.R7_Kreislauf_ohne_aussen,
           Typ                      := 0,
           FBa                      := #xTmp,
           FBa2                     := #xTmp,
           Out                      := Q     56.3);

NETWORK
TITLE =R7_Kreislauf_mit_aussen  Prog.schritt 16 CIP Krsl.m.ausse.
// Act 007
// Box           : FRM-A7
// Output address: Q56.4
      CALL FC    70 (
           UnitNo                   := #UnitNo,
           ActRec                   := DB2670.R7_Kreislauf_mit_aussen,
           Typ                      := 0,
           FBa                      := #xTmp,
           FBa2                     := #xTmp,
           Out                      := Q     56.4);

NETWORK
TITLE =R7_Grundstellung  Prog.schritt 1 Grundstellung
// Act 008
// Box           : FRM-A7
// Output address: Q56.2
      CALL FC    70 (
           UnitNo                   := #UnitNo,
           ActRec                   := DB2670.R7_Grundstellung,
           Typ                      := 0,
           FBa                      := #xTmp,
           FBa2                     := #xTmp,
           Out                      := Q     56.2);

NETWORK
TITLE =R7_Drainagestellung  Prog.schritt 2 Drainagestellung
// Act 009
// Box           : FRM-A7
// Output address: Q56.5
      CALL FC    70 (
           UnitNo                   := #UnitNo,
           ActRec                   := DB2670.R7_Drainagestellung,
           Typ                      := 0,
           FBa                      := #xTmp,
           FBa2                     := #xTmp,
           Out                      := Q     56.5);

NETWORK
TITLE =F7_Kreislauf_o_puls  Prog.schritt 15 CIP Krsl.o.ausse.
// Act 010
// Box           : FRM-A7
// Output address: Q54.2
      CALL FC    70 (
           UnitNo                   := #UnitNo,
           ActRec                   := DB2670.F7_Kreislauf_o_puls,
           Typ                      := 0,
           FBa                      := #xTmp,
           FBa2                     := #xTmp,
           Out                      := Q     54.2);

NETWORK
TITLE =F7_Kreislauf_m_puls  Prog.schritt 16 CIP Krsl.m.ausse.
// Act 011
// Box           : FRM-A7
// Output address: Q54.3
      CALL FC    70 (
           UnitNo                   := #UnitNo,
           ActRec                   := DB2670.F7_Kreislauf_m_puls,
           Typ                      := 0,
           FBa                      := #xTmp,
           FBa2                     := #xTmp,
           Out                      := Q     54.3);

NETWORK
TITLE =F7_Randvollstellung  Prog.schritt 17 Randv./Standdes.
// Act 012
// Box           : FRM-A7
// Output address: Q54.4
      CALL FC    70 (
           UnitNo                   := #UnitNo,
           ActRec                   := DB2670.F7_Randvollstellung,
           Typ                      := 0,
           FBa                      := #xTmp,
           FBa2                     := #xTmp,
           Out                      := Q     54.4);

NETWORK
TITLE =F7_Klarspuelen_o_CIP_Beh  Prog.schritt 19 Klarsp.o.CIP Beh
// Act 013
// Box           : FRM-A7
// Output address: Q54.5
      CALL FC    70 (
           UnitNo                   := #UnitNo,
           ActRec                   := DB2670.F7_Klarspuelen_o_CIP_Beh,
           Typ                      := 0,
           FBa                      := #xTmp,
           FBa2                     := #xTmp,
           Out                      := Q     54.5);

NETWORK
TITLE =F7_Ausschub_m_Sterilluft  Prog.schritt 20 Ausschub m.Steri
// Act 014
// Box           : FRM-A7
// Output address: Q54.6
      CALL FC    70 (
           UnitNo                   := #UnitNo,
           ActRec                   := DB2670.F7_Ausschub_m_Sterilluft,
           Typ                      := 0,
           FBa                      := #xTmp,
           FBa2                     := #xTmp,
           Out                      := Q     54.6);

NETWORK
TITLE =F7_Ausschub_m_CO2  Prog.schritt 21 Ausschub m.CO2
// Act 015
// Box           : FRM-A7
// Output address: Q54.7
      CALL FC    70 (
           UnitNo                   := #UnitNo,
           ActRec                   := DB2670.F7_Ausschub_m_CO2,
           Typ                      := 0,
           FBa                      := #xTmp,
           FBa2                     := #xTmp,
           Out                      := Q     54.7);

NETWORK
TITLE =F7_Grundstellung  Prog.schritt 1 Grundstellung
// Act 016
// Box           : FRM-A7
// Output address: Q55.0
      CALL FC    70 (
           UnitNo                   := #UnitNo,
           ActRec                   := DB2670.F7_Grundstellung,
           Typ                      := 0,
           FBa                      := #xTmp,
           FBa2                     := #xTmp,
           Out                      := Q     55.0);

NETWORK
TITLE =F7_Drainagestellung  Prog.schritt 2 Drainagestellung
// Act 017
// Box           : FRM-A7
// Output address: Q55.1
      CALL FC    70 (
           UnitNo                   := #UnitNo,
           ActRec                   := DB2670.F7_Drainagestellung,
           Typ                      := 0,
           FBa                      := #xTmp,
           FBa2                     := #xTmp,
           Out                      := Q     55.1);

NETWORK
TITLE =F7_Bypass  Prog.schritt 30 Bypass
// Act 018
// Box           : FRM-A7
// Output address: Q55.2
      CALL FC    70 (
           UnitNo                   := #UnitNo,
           ActRec                   := DB2670.F7_Bypass,
           Typ                      := 0,
           FBa                      := #xTmp,
           FBa2                     := #xTmp,
           Out                      := Q     55.2);

NETWORK
TITLE =A7_RR1  A7RR1 Ventil CIP Rücklauf Kreis 1 Anlage 7
// Act 020
// Box           : VSRR6-11
// Input address : I28.0
// Output address: Q28.0
      CALL FC    70 (
           UnitNo                   := #UnitNo,
           ActRec                   := DB2670.A7_RR1,
           Typ                      := 1,
           FBa                      := #xTmp,
           FBa2                     := I     28.0,
           Out                      := Q     28.0);

NETWORK
TITLE =A7_RR2  A7RR2 Ventil CIP Rücklauf Kreis 2 Anlage 7
// Act 021
// Box           : VSRR6-11
// Input address : I28.1
// Output address: Q28.1
      CALL FC    70 (
           UnitNo                   := #UnitNo,
           ActRec                   := DB2670.A7_RR2,
           Typ                      := 1,
           FBa                      := #xTmp,
           FBa2                     := I     28.1,
           Out                      := Q     28.1);

NETWORK
TITLE =A7_RR3  A7RR3 Ventil CIP Rücklauf Kreis 3 Anlage 7
// Act 022
// Box           : VSRR6-11
// Input address : I28.2
// Output address: Q28.2
      CALL FC    70 (
           UnitNo                   := #UnitNo,
           ActRec                   := DB2670.A7_RR3,
           Typ                      := 1,
           FBa                      := #xTmp,
           FBa2                     := I     28.2,
           Out                      := Q     28.2);

NETWORK
TITLE =M7_Grundstellung  Prog.schritt 101 Grundstellung
// Act 023
// Box           : FRM-A7
// Output address: Q58.0
      CALL FC    70 (
           UnitNo                   := #UnitNo,
           ActRec                   := DB2670.M7_Grundstellung,
           Typ                      := 0,
           FBa                      := #xTmp,
           FBa2                     := #xTmp,
           Out                      := Q     58.0);

NETWORK
TITLE =M7_Drainagestellung  Prog.schritt 102 Darinage
// Act 024
// Box           : FRM-A7
// Output address: Q58.1
      CALL FC    70 (
           UnitNo                   := #UnitNo,
           ActRec                   := DB2670.M7_Drainagestellung,
           Typ                      := 0,
           FBa                      := #xTmp,
           FBa2                     := #xTmp,
           Out                      := Q     58.1);

NETWORK
TITLE =M7_Ausspritzen_o_Ablauf  Prog.schritt 113 Ausspr.o.Ablauf
// Act 025
// Box           : FRM-A7
// Output address: Q58.2
      CALL FC    70 (
           UnitNo                   := #UnitNo,
           ActRec                   := DB2670.M7_Ausspritzen_o_Ablauf,
           Typ                      := 0,
           FBa                      := #xTmp,
           FBa2                     := #xTmp,
           Out                      := Q     58.2);

NETWORK
TITLE =M7_Ausspritzen_m_Ablauf  Prog.schritt 114 Ausspr.m.Ablauf
// Act 026
// Box           : FRM-A7
// Output address: Q58.3
      CALL FC    70 (
           UnitNo                   := #UnitNo,
           ActRec                   := DB2670.M7_Ausspritzen_m_Ablauf,
           Typ                      := 0,
           FBa                      := #xTmp,
           FBa2                     := #xTmp,
           Out                      := Q     58.3);

NETWORK
TITLE =M7_Fluten_o_Ablauf  Prog.schritt 115 Fluten o.Ablauf
// Act 027
// Box           : FRM-A7
// Output address: Q58.4
      CALL FC    70 (
           UnitNo                   := #UnitNo,
           ActRec                   := DB2670.M7_Fluten_o_Ablauf,
           Typ                      := 0,
           FBa                      := #xTmp,
           FBa2                     := #xTmp,
           Out                      := Q     58.4);

NETWORK
TITLE =M7_Fluten_m_Ablauf  Prog.schritt 116 Fluten m.Ablauf
// Act 028
// Box           : FRM-A7
// Output address: Q58.5
      CALL FC    70 (
           UnitNo                   := #UnitNo,
           ActRec                   := DB2670.M7_Fluten_m_Ablauf,
           Typ                      := 0,
           FBa                      := #xTmp,
           FBa2                     := #xTmp,
           Out                      := Q     58.5);

NETWORK
TITLE =M7_Randvollstellung  Prog.schritt 117 Randvollstellung
// Act 029
// Box           : FRM-A7
// Output address: Q58.6
      CALL FC    70 (
           UnitNo                   := #UnitNo,
           ActRec                   := DB2670.M7_Randvollstellung,
           Typ                      := 0,
           FBa                      := #xTmp,
           FBa2                     := #xTmp,
           Out                      := Q     58.6);

NETWORK
TITLE =M7_Abpumpen  Prog.schritt 118 Abpumpen
// Act 030
// Box           : FRM-A7
// Output address: Q58.7
      CALL FC    70 (
           UnitNo                   := #UnitNo,
           ActRec                   := DB2670.M7_Abpumpen,
           Typ                      := 0,
           FBa                      := #xTmp,
           FBa2                     := #xTmp,
           Out                      := Q     58.7);

NETWORK
TITLE =M7_Klarspuelen  Prog.schritt 119 Klarspuelen
// Act 031
// Box           : FRM-A7
// Output address: Q59.0
      CALL FC    70 (
           UnitNo                   := #UnitNo,
           ActRec                   := DB2670.M7_Klarspuelen,
           Typ                      := 0,
           FBa                      := #xTmp,
           FBa2                     := #xTmp,
           Out                      := Q     59.0);

END_FUNCTION_BLOCK

FUNCTION_BLOCK FB 1671
TITLE =U067: Packaging Plant 7
FAMILY : BOTEC_F1
NAME : UniE
VERSION : 1.2


VAR_TEMP
  CIP : BOOL ;	//CIP active
  UNIM : BOOL ;	//Unit Not In Maintenance
  GenRel : BOOL ;	//general OK (emergency and maintenance OK)
  EStopOK : BOOL ;	//emergency OK
  UnitNo : INT ;	//unit number
  xTmp : BOOL ;	//Temporary Bool
  iTmp : INT ;	//Temporary INT
  rTmp : REAL ;	//Temporary REAL
  dTmp : DINT ;	//Temporary DINT (free for general use)
  RetValInt : INT ;	//return value
END_VAR
BEGIN
NETWORK
TITLE =General

      SET   ;
// Simulation ---------------------------------------------------------------
      A     DB1671.DBX 1357.7;
      CC    FB  1679; // "U067Sim"
      A     DB1671.DBX   17.3;
      =     DB1671.DBX 1357.7; //Help bit for simulation

// get unit number ----------------------------------------------------------
      L     DB1670.DBW    0;
      T     #UnitNo;

// CIP ----------------------------------------------------------------------
      L     DB1671.DBD   54;
      L     0;
      <D    ;
      =     #CIP;

// emergency OK -------------------------------------------------------------
      A     DB1675.DBX   27.0; //Emergency Stop OK
      =     #EStopOK;

// Write Unit in Maintenance ------------------------------------------------

      AN    DB1671.DBX   69.7;
      =     #UNIM;

// emergency and maintenance OK ---------------------------------------------
      A     #EStopOK;
      A     #UNIM;
      =     #GenRel;

// communication ------------------------------------------------------------
      UC    FB  1675; // U067Com

NETWORK
TITLE =Universal Value

      NOP   0;

// ----------------------------------------------------------
// unv001 Process Status
// ----------------------------------------------------------
// process value to UnV
//      L     0.000000e+000
//      T     "U067UnVD".unv001.ValExt

// ----------------------------------------------------------
// unv002 Universal Value 02
// ----------------------------------------------------------
// process value to UnV
//      L     0.000000e+000
//      T     "U067UnVD".unv002.ValExt

// ----------------------------------------------------------
// unv003 Universal Value 03
// ----------------------------------------------------------
// process value to UnV
//      L     0.000000e+000
//      T     "U067UnVD".unv003.ValExt

// ----------------------------------------------------------
// unv004 Universal Value 04
// ----------------------------------------------------------
// process value to UnV
//      L     0.000000e+000
//      T     "U067UnVD".unv004.ValExt

NETWORK
TITLE =Special Input

      NOP   0;

// ----------------------------------------------------------
// A7_FUELLER_LAEUFT Fueller 7 laeuft
// ----------------------------------------------------------
//      CLR
//      =     "U067SpID".A7_FUELLER_LAEUFT.EAl
//      =     "U067SpID".A7_FUELLER_LAEUFT.Pre

// ----------------------------------------------------------
// A7_MIXER_CIP_BEREIT Mixer Anlage 7 CIP-Bereit
// ----------------------------------------------------------
//      A     #CIP
//      =     "U067SpID".A7_MIXER_CIP_BEREIT.EAl
//      =     "U067SpID".A7_MIXER_CIP_BEREIT.Pre

// ----------------------------------------------------------
// A7_MIXER_VOLL Mixer Anlage 7 voll
// ----------------------------------------------------------
//      CLR
//      =     "U067SpID".A7_MIXER_VOLL.EAl
//      =     "U067SpID".A7_MIXER_VOLL.Pre

// ----------------------------------------------------------
// A7_MIXER_LEER Mixer Anlage 7 leer
// ----------------------------------------------------------
//      CLR
//      =     "U067SpID".A7_MIXER_LEER.EAl
//      =     "U067SpID".A7_MIXER_LEER.Pre

// ----------------------------------------------------------
// A7_MIXER_ANF_SIRUP Mixer Anlage 7 Anforderung Sirup
// ----------------------------------------------------------
//      CLR
//      =     "U067SpID".A7_MIXER_ANF_SIRUP.EAl
//      =     "U067SpID".A7_MIXER_ANF_SIRUP.Pre

// ----------------------------------------------------------
// A7_SS_FRG_MOLCH Anlage 7 Schlüsselschalter Freigabe Molch
// ----------------------------------------------------------
//      CLR
//      =     "U067SpID".A7_SS_FRG_MOLCH.EAl
//      =     "U067SpID".A7_SS_FRG_MOLCH.Pre

// ----------------------------------------------------------
// A7_FUELLER_CIP_BEREIT Fueller 7 CIP-Bereit
// ----------------------------------------------------------
//      A     #CIP
//      =     "U067SpID".A7_FUELLER_CIP_BEREIT.EAl
//      =     "U067SpID".A7_FUELLER_CIP_BEREIT.Pre

// ----------------------------------------------------------
// A7_FUELLER_LEER Fueller 7 leer (Impuls)
// ----------------------------------------------------------
//      CLR
//      =     "U067SpID".A7_FUELLER_LEER.EAl
//      =     "U067SpID".A7_FUELLER_LEER.Pre

// ----------------------------------------------------------
// A7_RINSER_CIP_BEREIT Rinser Anlage 7 CIP-Bereit
// ----------------------------------------------------------
//      A     #CIP
//      =     "U067SpID".A7_RINSER_CIP_BEREIT.EAl
//      =     "U067SpID".A7_RINSER_CIP_BEREIT.Pre

// ----------------------------------------------------------
// A7_RINSER_LAEUFT Rinser Anlage 7 laeuft
// ----------------------------------------------------------
//      CLR
//      =     "U067SpID".A7_RINSER_LAEUFT.EAl
//      =     "U067SpID".A7_RINSER_LAEUFT.Pre

// ----------------------------------------------------------
// EA7_K1_Handklappe Handklappe Fueller 7
// ----------------------------------------------------------
//      CLR
//      =     "U067SpID".EA7_K1_Handklappe.EAl
//      =     "U067SpID".EA7_K1_Handklappe.Pre

NETWORK
TITLE =Messages

      NOP   0;

// ----------------------------------------------------------
// msg001 Message 01
// ----------------------------------------------------------
      SET   ;
      R     DB2677.DBX   80.7;
      =     DB2677.DBX   81.4;

      CLR   ;
      =     DB2677.DBX   82.7;

// ----------------------------------------------------------
// msg002 Message 02
// ----------------------------------------------------------
      SET   ;
      R     DB2677.DBX  140.7;
      =     DB2677.DBX  141.4;

      CLR   ;
      =     DB2677.DBX  142.7;

// ----------------------------------------------------------
// msg003 Message 03
// ----------------------------------------------------------
      SET   ;
      R     DB2677.DBX  200.7;
      =     DB2677.DBX  201.4;

      CLR   ;
      =     DB2677.DBX  202.7;

NETWORK
TITLE =Sequence organisation

      CLR   ;
      =     M    122.2;

// SFM supply ----------------------------------------------------------------

// sequencer ----------------------------------------------------------------
      A     DB1673.DBX   43.1;
      S     DB1673.DBX   97.3;

      CALL FC    40 (
           UnitNo                   := #UnitNo);

NETWORK
TITLE =Auto / Manual

      SET   ;
      AN    M    122.2;
      JC    MODE;
      AN    M    120.1;

// assign actuator mode
      AN    M    120.1;
      =     DB2670.DBX  105.4;
      =     DB2670.DBX  185.4;
      S     DB2670.DBX  265.4;
      =     DB2670.DBX  345.4;
      S     DB2670.DBX  425.4;
      =     DB2670.DBX  505.4;
      =     DB2670.DBX  585.4;
      =     DB2670.DBX  665.4;
      =     DB2670.DBX  745.4;
      =     DB2670.DBX  825.4;
      =     DB2670.DBX  905.4;
      =     DB2670.DBX  985.4;
      =     DB2670.DBX 1065.4;
      =     DB2670.DBX 1145.4;
      =     DB2670.DBX 1225.4;
      =     DB2670.DBX 1305.4;
      =     DB2670.DBX 1385.4;
      =     DB2670.DBX 1465.4;
      =     DB2670.DBX 1625.4;
      =     DB2670.DBX 1705.4;
      =     DB2670.DBX 1785.4;

      =     DB2670.DBX 1865.4;
      =     DB2670.DBX 1945.4;
      =     DB2670.DBX 2025.4;
      =     DB2670.DBX 2105.4;
      =     DB2670.DBX 2185.4;
      =     DB2670.DBX 2265.4;
      =     DB2670.DBX 2345.4;
      =     DB2670.DBX 2425.4;
      =     DB2670.DBX 2505.4;




MODE: SET   ;

NETWORK
TITLE =A7_RRP1 CIP Rücklaufpumpe Anlage 7
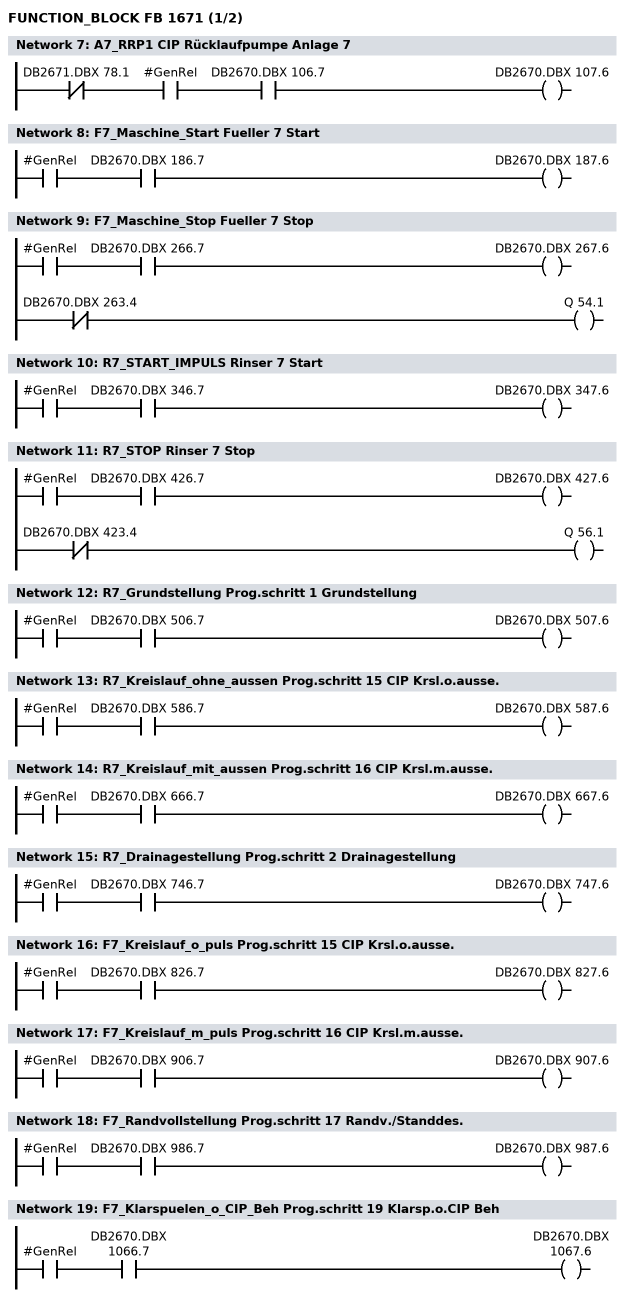

//      A     "U067SpID".FS_A7FS1.Sig
      AN    DB2671.DBX   78.1;

      A     #GenRel;
      A     DB2670.DBX  106.7;
      =     DB2670.DBX  107.6;
NETWORK
TITLE =F7_Maschine_Start Fueller 7 Start

      A     #GenRel;
      A     DB2670.DBX  186.7;
      =     DB2670.DBX  187.6;
NETWORK
TITLE =F7_Maschine_Stop Fueller 7 Stop

      A     #GenRel;
      A     DB2670.DBX  266.7;
      =     DB2670.DBX  267.6;

      AN    DB2670.DBX  263.4;
      =     Q     54.1;
NETWORK
TITLE =R7_START_IMPULS Rinser 7 Start

      A     #GenRel;
      A     DB2670.DBX  346.7;
      =     DB2670.DBX  347.6;


NETWORK
TITLE =R7_STOP Rinser 7 Stop

      A     #GenRel;
      A     DB2670.DBX  426.7;
      =     DB2670.DBX  427.6;

      AN    DB2670.DBX  423.4;
      =     Q     56.1;

NETWORK
TITLE =R7_Grundstellung Prog.schritt 1 Grundstellung

      A     #GenRel;
      A     DB2670.DBX  506.7;
      =     DB2670.DBX  507.6;
NETWORK
TITLE =R7_Kreislauf_ohne_aussen Prog.schritt 15 CIP Krsl.o.ausse.

      A     #GenRel;
      A     DB2670.DBX  586.7;
      =     DB2670.DBX  587.6;
NETWORK
TITLE =R7_Kreislauf_mit_aussen Prog.schritt 16 CIP Krsl.m.ausse.

      A     #GenRel;
      A     DB2670.DBX  666.7;
      =     DB2670.DBX  667.6;
NETWORK
TITLE =R7_Drainagestellung Prog.schritt 2 Drainagestellung

      A     #GenRel;
      A     DB2670.DBX  746.7;
      =     DB2670.DBX  747.6;
NETWORK
TITLE =F7_Kreislauf_o_puls Prog.schritt 15 CIP Krsl.o.ausse.

      A     #GenRel;
      A     DB2670.DBX  826.7;
      =     DB2670.DBX  827.6;
NETWORK
TITLE =F7_Kreislauf_m_puls Prog.schritt 16 CIP Krsl.m.ausse.

      A     #GenRel;
      A     DB2670.DBX  906.7;
      =     DB2670.DBX  907.6;
NETWORK
TITLE =F7_Randvollstellung Prog.schritt 17 Randv./Standdes.

      A     #GenRel;
      A     DB2670.DBX  986.7;
      =     DB2670.DBX  987.6;
NETWORK
TITLE =F7_Klarspuelen_o_CIP_Beh Prog.schritt 19 Klarsp.o.CIP Beh

      A     #GenRel;
      A     DB2670.DBX 1066.7;
      =     DB2670.DBX 1067.6;
NETWORK
TITLE =F7_Ausschub_m_Sterilluft Prog.schritt 20 Ausschub m.Steri
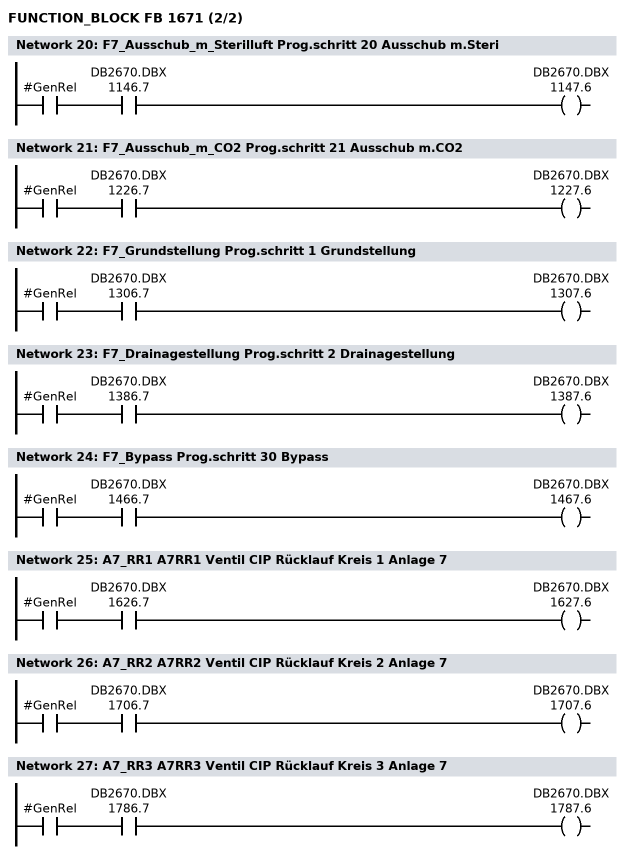

      A     #GenRel;
      A     DB2670.DBX 1146.7;
      =     DB2670.DBX 1147.6;
NETWORK
TITLE =F7_Ausschub_m_CO2 Prog.schritt 21 Ausschub m.CO2

      A     #GenRel;
      A     DB2670.DBX 1226.7;
      =     DB2670.DBX 1227.6;
NETWORK
TITLE =F7_Grundstellung Prog.schritt 1 Grundstellung

      A     #GenRel;
      A     DB2670.DBX 1306.7;
      =     DB2670.DBX 1307.6;
NETWORK
TITLE =F7_Drainagestellung Prog.schritt 2 Drainagestellung

      A     #GenRel;
      A     DB2670.DBX 1386.7;
      =     DB2670.DBX 1387.6;
NETWORK
TITLE =F7_Bypass Prog.schritt 30 Bypass

      A     #GenRel;
      A     DB2670.DBX 1466.7;
      =     DB2670.DBX 1467.6;
NETWORK
TITLE =A7_RR1 A7RR1 Ventil CIP Rücklauf Kreis 1 Anlage 7

      A     #GenRel;
      A     DB2670.DBX 1626.7;
      =     DB2670.DBX 1627.6;
NETWORK
TITLE =A7_RR2 A7RR2 Ventil CIP Rücklauf Kreis 2 Anlage 7

      A     #GenRel;
      A     DB2670.DBX 1706.7;
      =     DB2670.DBX 1707.6;
NETWORK
TITLE =A7_RR3 A7RR3 Ventil CIP Rücklauf Kreis 3 Anlage 7

      A     #GenRel;
      A     DB2670.DBX 1786.7;
      =     DB2670.DBX 1787.6;
END_FUNCTION_BLOCK

FUNCTION_BLOCK FB 1680
TITLE =U068: Packaging Plant 8
FAMILY : BOTEC_F1
NAME : UniA
VERSION : 2.1


VAR_TEMP
  EStopOK : BOOL ;	//auxiliary flag
  CIP : BOOL ;	//CIP Program Selected
  xTmp : BOOL ;	//Temporary Bool(free for general use)
  UnitNo : INT ;	//unit number
  UnitFB : INT ;	//unit expansion FB number
  rTmp : REAL ;	//Temporary REAL (free for general use)
  iTmp : INT ;	//Temporary INT (free for general use)
  dTmp : DINT ;	//Temporary DINT (free for general use)
END_VAR
BEGIN
NETWORK
TITLE =general

      CLR   ;
      =     #xTmp;
      =     #EStopOK;

      L     DB1680.DBW    0;
      T     #UnitNo;
      L     DB1680.DBW    2;
      T     #UnitFB;

NETWORK
TITLE =Universal value

      NOP   0;
// unv001 UnV 001 Process Status
      CALL FC    27 (
           UnitNo                   := #UnitNo,
           UnVRec                   := DB2685.unv001,
           ValExt                   := DB2685.DBD  234);

// unv002 UnV 002 Universal Value 02
      CALL FC    27 (
           UnitNo                   := #UnitNo,
           UnVRec                   := DB2685.unv002,
           ValExt                   := DB2685.DBD  362);

// unv003 UnV 003 Universal Value 03
      CALL FC    27 (
           UnitNo                   := #UnitNo,
           UnVRec                   := DB2685.unv003,
           ValExt                   := DB2685.DBD  490);

// unv004 UnV 004 Universal Value 04
      CALL FC    27 (
           UnitNo                   := #UnitNo,
           UnVRec                   := DB2685.unv004,
           ValExt                   := DB2685.DBD  618);

NETWORK
TITLE =special inputs

      NOP   0;
// DT_STOP_FUELLER_8 SpI 002 Anlage 8 Taster STOP
      CALL FC    14 (
           UnitNo                   := #UnitNo,
           SpIRec                   := DB2681.DT_STOP_FUELLER_8,
           SpIBit                   := I    113.4);

// DT_START_FUELLER_8 SpI 003 Anlage 8 Taster START
      CALL FC    14 (
           UnitNo                   := #UnitNo,
           SpIRec                   := DB2681.DT_START_FUELLER_8,
           SpIBit                   := I    113.5);

// A8_LAMPENTEST SpI 011 Anlage 8 Taster Lampen prüfen
      CALL FC    14 (
           UnitNo                   := #UnitNo,
           SpIRec                   := DB2681.A8_LAMPENTEST,
           SpIBit                   := I    112.7);

// A8_A8V1_HAND SpI 024 Anlage 8 Schalter Handansteuerung Ventil A8V1
      CALL FC    14 (
           UnitNo                   := #UnitNo,
           SpIRec                   := DB2681.A8_A8V1_HAND,
           SpIBit                   := I    113.0);

// A8_A8V2_HAND SpI 025 Anlage 8 Schalter Handansteuerung Ventil A8V2
      CALL FC    14 (
           UnitNo                   := #UnitNo,
           SpIRec                   := DB2681.A8_A8V2_HAND,
           SpIBit                   := I    113.1);

// A8_A8V3_HAND SpI 026 Anlage 8 Schalter Handansteuerung Ventil A8V3
      CALL FC    14 (
           UnitNo                   := #UnitNo,
           SpIRec                   := DB2681.A8_A8V3_HAND,
           SpIBit                   := I    113.2);

// A8_ANFORD_WASSER SpI 027 Anlage 8 Schalter Anforderung Wasser (RWPA8)
      CALL FC    14 (
           UnitNo                   := #UnitNo,
           SpIRec                   := DB2681.A8_ANFORD_WASSER,
           SpIBit                   := I    113.3);

// A8_SS_HAND SpI 028 Anlage 8 Schlüsselschalter Hand
      CALL FC    14 (
           UnitNo                   := #UnitNo,
           SpIRec                   := DB2681.A8_SS_HAND,
           SpIBit                   := I    113.6);

NETWORK
TITLE =messages

      NOP   0;
// msg001 Msg 001 Message 01
      CALL FC    16 (
           UnitNo                   := #UnitNo,
           MsgRec                   := DB2687.msg001,
           MsgBit                   := DB2687.DBX   82.7);

// msg002 Msg 002 Message 02
      CALL FC    16 (
           UnitNo                   := #UnitNo,
           MsgRec                   := DB2687.msg002,
           MsgBit                   := DB2687.DBX  142.7);

// msg003 Msg 003 Message 03
      CALL FC    16 (
           UnitNo                   := #UnitNo,
           MsgRec                   := DB2687.msg003,
           MsgBit                   := DB2687.DBX  202.7);

NETWORK
TITLE =unit supply

      UC    FB [#UnitFB];

NETWORK
TITLE =RWP_A8  RWPA8 Anlage 8 Befüllpumpe
// Act 001
// Box           : VSA8
// Input address : I112.3
// Output address: Q44.3
      CALL FC    70 (
           UnitNo                   := #UnitNo,
           ActRec                   := DB2680.RWP_A8,
           Typ                      := 3,
           FBa                      := I    112.3,
           FBa2                     := #xTmp,
           Out                      := Q     44.3);

NETWORK
TITLE =A8_V1  A8V1 Anlage 8 Ventil Filter
// Act 002
// Box           : VSA8
// Input address : I112.0
// Output address: Q44.0
      CALL FC    70 (
           UnitNo                   := #UnitNo,
           ActRec                   := DB2680.A8_V1,
           Typ                      := 0,
           FBa                      := #xTmp,
           FBa2                     := I    112.0,
           Out                      := Q     44.0);

NETWORK
TITLE =A8_V2  A8V2 Anlage 8 Ventil Filter
// Act 003
// Box           : VSA8
// Input address : I112.1
// Output address: Q44.1
      CALL FC    70 (
           UnitNo                   := #UnitNo,
           ActRec                   := DB2680.A8_V2,
           Typ                      := 0,
           FBa                      := #xTmp,
           FBa2                     := I    112.1,
           Out                      := Q     44.1);

NETWORK
TITLE =A8_V3  A8V3 Anlage 8 Ventil Filter
// Act 004
// Box           : VSA8
// Input address : I112.2
// Output address: Q44.2
      CALL FC    70 (
           UnitNo                   := #UnitNo,
           ActRec                   := DB2680.A8_V3,
           Typ                      := 0,
           FBa                      := #xTmp,
           FBa2                     := I    112.2,
           Out                      := Q     44.2);

NETWORK
TITLE =LA_A8_V1  Anlage 8 Lampe A8V1
// Act 005
// Box           : VSA8
// Output address: Q45.0
      CALL FC    70 (
           UnitNo                   := #UnitNo,
           ActRec                   := DB2680.LA_A8_V1,
           Typ                      := 0,
           FBa                      := #xTmp,
           FBa2                     := #xTmp,
           Out                      := Q     45.0);

NETWORK
TITLE =LA_A8_V2  Anlage 8 Lampe A8V2
// Act 006
// Box           : VSA8
// Output address: Q45.1
      CALL FC    70 (
           UnitNo                   := #UnitNo,
           ActRec                   := DB2680.LA_A8_V2,
           Typ                      := 0,
           FBa                      := #xTmp,
           FBa2                     := #xTmp,
           Out                      := Q     45.1);

NETWORK
TITLE =LA_A8_V3  Anlage 8 Lampe A8V3
// Act 007
// Box           : VSA8
// Output address: Q45.2
      CALL FC    70 (
           UnitNo                   := #UnitNo,
           ActRec                   := DB2680.LA_A8_V3,
           Typ                      := 0,
           FBa                      := #xTmp,
           FBa2                     := #xTmp,
           Out                      := Q     45.2);

NETWORK
TITLE =LA_A8_RWPA8  Anlage 8 Lampe RWPA8
// Act 008
// Box           : VSA8
// Output address: Q45.3
      CALL FC    70 (
           UnitNo                   := #UnitNo,
           ActRec                   := DB2680.LA_A8_RWPA8,
           Typ                      := 0,
           FBa                      := #xTmp,
           FBa2                     := #xTmp,
           Out                      := Q     45.3);

NETWORK
TITLE =LA_A8_PROD  Anlage 8 Lampe Produktion
// Act 009
// Box           : VSA8
// Output address: Q45.6
      CALL FC    70 (
           UnitNo                   := #UnitNo,
           ActRec                   := DB2680.LA_A8_PROD,
           Typ                      := 0,
           FBa                      := #xTmp,
           FBa2                     := #xTmp,
           Out                      := Q     45.6);

NETWORK
TITLE =LA_A8_CIP  Anlage 8 Lampe CIP
// Act 010
// Box           : VSA8
// Output address: Q45.7
      CALL FC    70 (
           UnitNo                   := #UnitNo,
           ActRec                   := DB2680.LA_A8_CIP,
           Typ                      := 0,
           FBa                      := #xTmp,
           FBa2                     := #xTmp,
           Out                      := Q     45.7);

NETWORK
TITLE =A8_RR1  A8RR1 CIP Rücklaufventil Kreis 1 Anlage 8
// Act 020
// Box           : VS-RRA
// Input address : I200.0
// Output address: Q200.0
      CALL FC    70 (
           UnitNo                   := #UnitNo,
           ActRec                   := DB2680.A8_RR1,
           Typ                      := 0,
           FBa                      := #xTmp,
           FBa2                     := I    200.0,
           Out                      := Q    200.0);

NETWORK
TITLE =A8_RR2  A8RR2 CIP Rücklaufventil Kreis 2 Anlage 8
// Act 021
// Box           : VS-RRA
// Input address : I200.1
// Output address: Q200.1
      CALL FC    70 (
           UnitNo                   := #UnitNo,
           ActRec                   := DB2680.A8_RR2,
           Typ                      := 0,
           FBa                      := #xTmp,
           FBa2                     := I    200.1,
           Out                      := Q    200.1);

NETWORK
TITLE =A8_RR3  A8RR3 CIP Rücklaufventil Kreis 3 Anlage 8
// Act 022
// Box           : VS-RRA
// Input address : I200.2
// Output address: Q200.2
      CALL FC    70 (
           UnitNo                   := #UnitNo,
           ActRec                   := DB2680.A8_RR3,
           Typ                      := 0,
           FBa                      := #xTmp,
           FBa2                     := I    200.2,
           Out                      := Q    200.2);

END_FUNCTION_BLOCK

FUNCTION_BLOCK FB 1681
TITLE =U068: Packaging Plant 8
FAMILY : BOTEC_F1
NAME : UniE
VERSION : 1.2


VAR_TEMP
  CIP : BOOL ;	//CIP active
  UNIM : BOOL ;	//Unit Not In Maintenance
  GenRel : BOOL ;	//general OK (emergency and maintenance OK)
  EStopOK : BOOL ;	//emergency OK
  UnitNo : INT ;	//unit number
  xTmp : BOOL ;	//Temporary Bool
  iTmp : INT ;	//Temporary INT
  rTmp : REAL ;	//Temporary REAL
  dTmp : DINT ;	//Temporary DINT (free for general use)
  RetValInt : INT ;	//return value
END_VAR
BEGIN
NETWORK
TITLE =General

      SET   ;
// Simulation ---------------------------------------------------------------
      A     DB1681.DBX 1357.7;
      CC    FB  1689; // "U068Sim"
      A     DB1681.DBX   17.3;
      =     DB1681.DBX 1357.7; //Help bit for simulation

// get unit number ----------------------------------------------------------
      L     DB1680.DBW    0;
      T     #UnitNo;

// CIP ----------------------------------------------------------------------
      L     DB1681.DBD   54;
      L     0;
      <D    ;
      =     #CIP;

// emergency OK -------------------------------------------------------------
      A     DB1685.DBX   27.0; //Emergency Stop OK
      =     #EStopOK;

// Write Unit in Maintenance ------------------------------------------------

      AN    DB1681.DBX   69.7;
      =     #UNIM;

// emergency and maintenance OK ---------------------------------------------
      A     #EStopOK;
      A     #UNIM;
      =     #GenRel;

// communication ------------------------------------------------------------
      UC    FB  1685; // U068Com

NETWORK
TITLE =Universal Value

      NOP   0;

// ----------------------------------------------------------
// unv001 Process Status
// ----------------------------------------------------------
// process value to UnV
//      L     0.000000e+000
//      T     "U068UnVD".unv001.ValExt

// ----------------------------------------------------------
// unv002 Universal Value 02
// ----------------------------------------------------------
// process value to UnV
//      L     0.000000e+000
//      T     "U068UnVD".unv002.ValExt

// ----------------------------------------------------------
// unv003 Universal Value 03
// ----------------------------------------------------------
// process value to UnV
//      L     0.000000e+000
//      T     "U068UnVD".unv003.ValExt

// ----------------------------------------------------------
// unv004 Universal Value 04
// ----------------------------------------------------------
// process value to UnV
//      L     0.000000e+000
//      T     "U068UnVD".unv004.ValExt

NETWORK
TITLE =Special Input

      NOP   0;

// ----------------------------------------------------------
// DT_STOP_FUELLER_8 Anlage 8 Taster STOP
// ----------------------------------------------------------
      CLR   ;
      =     DB2681.DBX  141.4;
      =     DB2681.DBX  141.5;

// ----------------------------------------------------------
// DT_START_FUELLER_8 Anlage 8 Taster START
// ----------------------------------------------------------
      CLR   ;
      =     DB2681.DBX  201.4;
      =     DB2681.DBX  201.5;

// ----------------------------------------------------------
// A8_LAMPENTEST Anlage 8 Taster Lampen prüfen
// ----------------------------------------------------------
      CLR   ;
      =     DB2681.DBX  681.4;
      =     DB2681.DBX  681.5;

// ----------------------------------------------------------
// A8_A8V1_HAND Anlage 8 Schalter Handansteuerung Ventil A8V1
// ----------------------------------------------------------
      CLR   ;
      =     DB2681.DBX 1461.4;
      =     DB2681.DBX 1461.5;

// ----------------------------------------------------------
// A8_A8V2_HAND Anlage 8 Schalter Handansteuerung Ventil A8V2
// ----------------------------------------------------------
      CLR   ;
      =     DB2681.DBX 1521.4;
      =     DB2681.DBX 1521.5;

// ----------------------------------------------------------
// A8_A8V3_HAND Anlage 8 Schalter Handansteuerung Ventil A8V3
// ----------------------------------------------------------
      CLR   ;
      =     DB2681.DBX 1581.4;
      =     DB2681.DBX 1581.5;

// ----------------------------------------------------------
// A8_ANFORD_WASSER Anlage 8 Schalter Anforderung Wasser (RWPA8)
// ----------------------------------------------------------
      CLR   ;
      =     DB2681.DBX 1641.4;
      =     DB2681.DBX 1641.5;

// ----------------------------------------------------------
// A8_SS_HAND Anlage 8 Schlüsselschalter Hand
// ----------------------------------------------------------
      CLR   ;
      =     DB2681.DBX 1701.4;
      =     DB2681.DBX 1701.5;

NETWORK
TITLE =Messages

      NOP   0;

// ----------------------------------------------------------
// msg001 Message 01
// ----------------------------------------------------------
      SET   ;
      R     DB2687.DBX   80.7;
      =     DB2687.DBX   81.4;

      CLR   ;
      =     DB2687.DBX   82.7;

// ----------------------------------------------------------
// msg002 Message 02
// ----------------------------------------------------------
      SET   ;
      R     DB2687.DBX  140.7;
      =     DB2687.DBX  141.4;

      CLR   ;
      =     DB2687.DBX  142.7;

// ----------------------------------------------------------
// msg003 Message 03
// ----------------------------------------------------------
      SET   ;
      R     DB2687.DBX  200.7;
      =     DB2687.DBX  201.4;

      CLR   ;
      =     DB2687.DBX  202.7;

NETWORK
TITLE =Sequence organisation

      CLR   ;
      =     M    122.2;

// SFM supply ----------------------------------------------------------------

// sequencer ----------------------------------------------------------------
      A     DB1683.DBX   43.1;
      S     DB1683.DBX   97.3;

      CALL FC    40 (
           UnitNo                   := #UnitNo);

NETWORK
TITLE =Auto / Manual

      SET   ;
      AN    M    122.2;
      JC    MODE;
      AN    M    120.1;

// assign actuator mode
      AN    M    120.1;
      =     DB2680.DBX  105.4;
      =     DB2680.DBX  185.4;
      =     DB2680.DBX  265.4;
      =     DB2680.DBX  345.4;
      =     DB2680.DBX  425.4;
      =     DB2680.DBX  505.4;
      =     DB2680.DBX  585.4;
      =     DB2680.DBX  665.4;
      =     DB2680.DBX  745.4;
      =     DB2680.DBX  825.4;
      =     DB2680.DBX 1625.4;
      =     DB2680.DBX 1705.4;
      =     DB2680.DBX 1785.4;



MODE: SET   ;

NETWORK
TITLE =RWP_A8 RWPA8 Anlage 8 Befüllpumpe
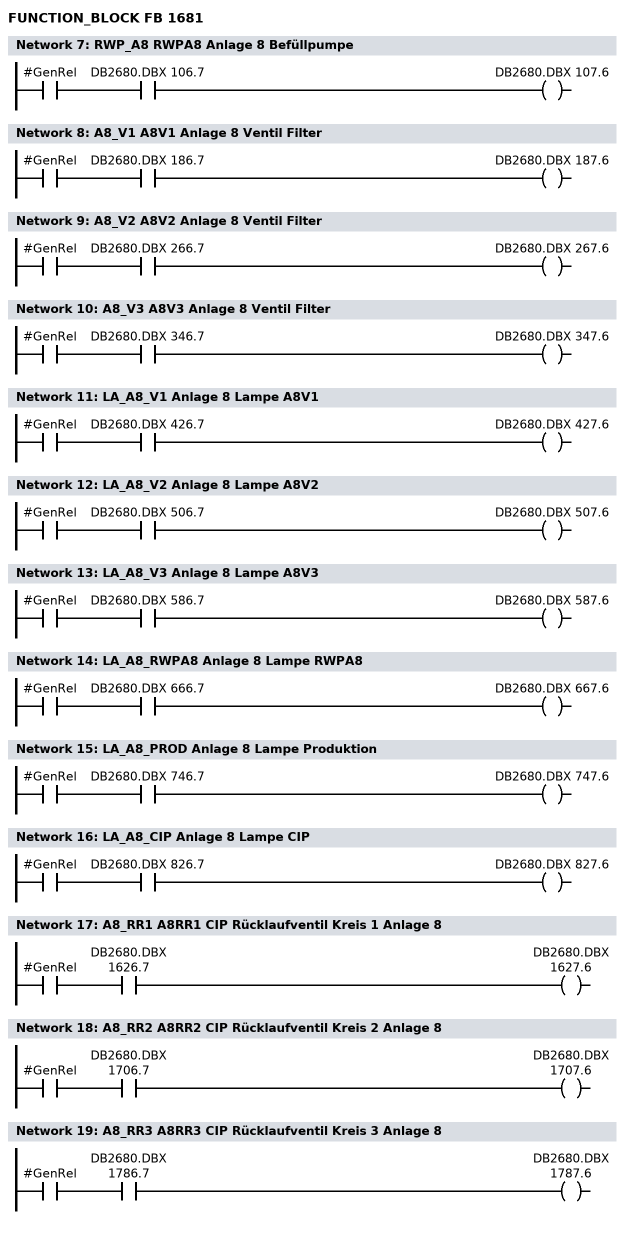

      A     #GenRel;
      A     DB2680.DBX  106.7;
      =     DB2680.DBX  107.6;
NETWORK
TITLE =A8_V1 A8V1 Anlage 8 Ventil Filter

      A     #GenRel;
      A     DB2680.DBX  186.7;
      =     DB2680.DBX  187.6;
NETWORK
TITLE =A8_V2 A8V2 Anlage 8 Ventil Filter

      A     #GenRel;
      A     DB2680.DBX  266.7;
      =     DB2680.DBX  267.6;
NETWORK
TITLE =A8_V3 A8V3 Anlage 8 Ventil Filter

      A     #GenRel;
      A     DB2680.DBX  346.7;
      =     DB2680.DBX  347.6;
NETWORK
TITLE =LA_A8_V1 Anlage 8 Lampe A8V1

      A     #GenRel;
      A     DB2680.DBX  426.7;
      =     DB2680.DBX  427.6;
NETWORK
TITLE =LA_A8_V2 Anlage 8 Lampe A8V2

      A     #GenRel;
      A     DB2680.DBX  506.7;
      =     DB2680.DBX  507.6;
NETWORK
TITLE =LA_A8_V3 Anlage 8 Lampe A8V3

      A     #GenRel;
      A     DB2680.DBX  586.7;
      =     DB2680.DBX  587.6;
NETWORK
TITLE =LA_A8_RWPA8 Anlage 8 Lampe RWPA8

      A     #GenRel;
      A     DB2680.DBX  666.7;
      =     DB2680.DBX  667.6;
NETWORK
TITLE =LA_A8_PROD Anlage 8 Lampe Produktion

      A     #GenRel;
      A     DB2680.DBX  746.7;
      =     DB2680.DBX  747.6;
NETWORK
TITLE =LA_A8_CIP Anlage 8 Lampe CIP

      A     #GenRel;
      A     DB2680.DBX  826.7;
      =     DB2680.DBX  827.6;
NETWORK
TITLE =A8_RR1 A8RR1 CIP Rücklaufventil Kreis 1 Anlage 8

      A     #GenRel;
      A     DB2680.DBX 1626.7;
      =     DB2680.DBX 1627.6;
NETWORK
TITLE =A8_RR2 A8RR2 CIP Rücklaufventil Kreis 2 Anlage 8

      A     #GenRel;
      A     DB2680.DBX 1706.7;
      =     DB2680.DBX 1707.6;
NETWORK
TITLE =A8_RR3 A8RR3 CIP Rücklaufventil Kreis 3 Anlage 8

      A     #GenRel;
      A     DB2680.DBX 1786.7;
      =     DB2680.DBX 1787.6;
END_FUNCTION_BLOCK

FUNCTION_BLOCK FB 1690
TITLE =U069: Abfüllanlage  9
FAMILY : BOTEC_F1
NAME : U069A
VERSION : 2.1


VAR_TEMP
  EStopOK : BOOL ;	//auxiliary flag
  CIP : BOOL ;	//CIP Program Selected
  xTmp : BOOL ;	//Temporary Bool(free for general use)
  DummyBool : BOOL ;	//Temporary Bool(free for general use)
  UnitNo : INT ;	//unit number
  UnitFB : INT ;	//unit expansion FB number
  rTmp : REAL ;	//Temporary REAL (free for general use)
  iTmp : INT ;	//Temporary INT (free for general use)
  DummyInt : INT ;	//Temporary INT (free for general use)
  dTmp : DINT ;	//Temporary DINT (free for general use)
END_VAR
BEGIN
NETWORK
TITLE =general

      CLR   ;
      =     #xTmp;
      =     #EStopOK;

      L     DB1690.DBW    0;
      T     #UnitNo;
      L     DB1690.DBW    2;
      T     #UnitFB;

NETWORK
TITLE =analog inputs

      NOP   0;
// HWWT1_TT01 AnI 001 Heißwasser-Wärmetauscher1 TT01
      CALL FC    24 (
           UnitNo                   := #UnitNo,
           AnIRec                   := DB2693.HWWT1_TT01,
           ValPer                   := PIW  236);

NETWORK
TITLE =Universal value

      NOP   0;
// unv001 UnV 001 Process Status
      CALL FC    27 (
           UnitNo                   := #UnitNo,
           UnVRec                   := DB2695.unv001,
           ValExt                   := DB2695.DBD  234);

// unv002 UnV 002 Universal Value 02
      CALL FC    27 (
           UnitNo                   := #UnitNo,
           UnVRec                   := DB2695.unv002,
           ValExt                   := DB2695.DBD  362);

// unv003 UnV 003 Universal Value 03
      CALL FC    27 (
           UnitNo                   := #UnitNo,
           UnVRec                   := DB2695.unv003,
           ValExt                   := DB2695.DBD  490);

// unv004 UnV 004 Universal Value 04
      CALL FC    27 (
           UnitNo                   := #UnitNo,
           UnVRec                   := DB2695.unv004,
           ValExt                   := DB2695.DBD  618);

NETWORK
TITLE =special inputs

      NOP   0;
// A9_FS1 SpI 001 geändert 07.11.01 A11 FS1 Stömungswächter
      CALL FC    14 (
           UnitNo                   := #UnitNo,
           SpIRec                   := DB2691.A9_FS1,
           SpIBit                   := I    177.0);

// TS_HL_ANL9 SpI 002
      CALL FC    14 (
           UnitNo                   := #UnitNo,
           SpIRec                   := DB2691.TS_HL_ANL9,
           SpIBit                   := I     62.0);

// GOA_903 SpI 004 geändert 07.11.01
      CALL FC    14 (
           UnitNo                   := #UnitNo,
           SpIRec                   := DB2691.GOA_903,
           SpIBit                   := I    176.2);

// LDT_A9_PRODUKT SpI 008 AB FUELLER 9/10
      CALL FC    14 (
           UnitNo                   := #UnitNo,
           SpIRec                   := DB2691.LDT_A9_PRODUKT,
           SpIBit                   := I     52.3);

// LDT_A9_CIP SpI 009 AB FUELLER 9/10
      CALL FC    14 (
           UnitNo                   := #UnitNo,
           SpIRec                   := DB2691.LDT_A9_CIP,
           SpIBit                   := I     52.4);

// DT_A9_START SpI 010 AB FUELLER 9/10
      CALL FC    14 (
           UnitNo                   := #UnitNo,
           SpIRec                   := DB2691.DT_A9_START,
           SpIBit                   := I     52.5);

// DT_A9_STOP SpI 011 AB FUELLER 9/10
      CALL FC    14 (
           UnitNo                   := #UnitNo,
           SpIRec                   := DB2691.DT_A9_STOP,
           SpIBit                   := I     52.6);

// DT_LAMPEN_PRUEFEN_A9_L10 SpI 012 AB FUELLER 9/10
      CALL FC    14 (
           UnitNo                   := #UnitNo,
           SpIRec                   := DB2691.DT_LAMPEN_PRUEFEN_A9_L10,
           SpIBit                   := I     53.6);

// QUITT_A9_LA10 SpI 013
      CALL FC    14 (
           UnitNo                   := #UnitNo,
           SpIRec                   := DB2691.QUITT_A9_LA10,
           SpIBit                   := I     53.7);

// BETRIEB_F9 SpI 014 SIGNAL VON FUELLER 9
      CALL FC    14 (
           UnitNo                   := #UnitNo,
           SpIRec                   := DB2691.BETRIEB_F9,
           SpIBit                   := I     62.4);

// BETRIEB_MIX_LKASKADE_F9 SpI 015 SIGNAL VON FUELLER 9
      CALL FC    14 (
           UnitNo                   := #UnitNo,
           SpIRec                   := DB2691.BETRIEB_MIX_LKASKADE_F9,
           SpIBit                   := I     62.6);

// M9_Produkt_kommt SpI 016 Meldung von Mixer9 für Heißabfüllung-Ausschub
      CALL FC    14 (
           UnitNo                   := #UnitNo,
           SpIRec                   := DB2691.M9_Produkt_kommt,
           SpIBit                   := I     40.7);

// F9_TEMPERATUR_ERREICHT SpI 017 SIGNAL VON FUELLER 9
      CALL FC    14 (
           UnitNo                   := #UnitNo,
           SpIRec                   := DB2691.F9_TEMPERATUR_ERREICHT,
           SpIBit                   := I     41.0);

// F9_TEMPERATUR_MIN_LMAX SpI 018 SIGNAL VON FUELLER 9
      CALL FC    14 (
           UnitNo                   := #UnitNo,
           SpIRec                   := DB2691.F9_TEMPERATUR_MIN_LMAX,
           SpIBit                   := I     41.1);

// F9_ANF_PRODUKTPUMPE SpI 019 SIGNAL VON FUELLER 9
      CALL FC    14 (
           UnitNo                   := #UnitNo,
           SpIRec                   := DB2691.F9_ANF_PRODUKTPUMPE,
           SpIBit                   := I     41.2);

// F9_PRODUKTIONSENDE SpI 020 SIGNAL VON FUELLER 9
      CALL FC    14 (
           UnitNo                   := #UnitNo,
           SpIRec                   := DB2691.F9_PRODUKTIONSENDE,
           SpIBit                   := I     41.3);

// F9_BETRIEBSBEREIT SpI 021 SIGNAL VON FUELLER 9
      CALL FC    14 (
           UnitNo                   := #UnitNo,
           SpIRec                   := DB2691.F9_BETRIEBSBEREIT,
           SpIBit                   := I     41.4);

// RM_RWPA9 SpI 022 SIGNAL VON MIXER F9/10
      CALL FC    14 (
           UnitNo                   := #UnitNo,
           SpIRec                   := DB2691.RM_RWPA9,
           SpIBit                   := I    122.5);

// MIX_WEGFREIGABE_9_L9 SpI 023 SIGNAL VON MIXER A9/10
      CALL FC    14 (
           UnitNo                   := #UnitNo,
           SpIRec                   := DB2691.MIX_WEGFREIGABE_9_L9,
           SpIBit                   := I    122.6);

// MIX_WEGFREIGABE_9_L10 SpI 024 SIGNAL VON MIXER A9/10
      CALL FC    14 (
           UnitNo                   := #UnitNo,
           SpIRec                   := DB2691.MIX_WEGFREIGABE_9_L10,
           SpIBit                   := I    122.7);

// MIX_ANFORDERUNG_PUMPE SpI 025 SIGNAL VON MIXER F9/F10
      CALL FC    14 (
           UnitNo                   := #UnitNo,
           SpIRec                   := DB2691.MIX_ANFORDERUNG_PUMPE,
           SpIBit                   := I    122.4);

// LS_LLL_A9 SpI 034 SIGNAL VON FUELLER 9
      CALL FC    14 (
           UnitNo                   := #UnitNo,
           SpIRec                   := DB2691.LS_LLL_A9,
           SpIBit                   := I     62.2);

NETWORK
TITLE =messages

      NOP   0;
// msg001 Msg 001 Message 01
      CALL FC    16 (
           UnitNo                   := #UnitNo,
           MsgRec                   := DB2697.msg001,
           MsgBit                   := DB2697.DBX   82.7);

// msg002 Msg 002 Message 02
      CALL FC    16 (
           UnitNo                   := #UnitNo,
           MsgRec                   := DB2697.msg002,
           MsgBit                   := DB2697.DBX  142.7);

// msg003 Msg 003 Message 03
      CALL FC    16 (
           UnitNo                   := #UnitNo,
           MsgRec                   := DB2697.msg003,
           MsgBit                   := DB2697.DBX  202.7);

NETWORK
TITLE =unit supply

      UC    FB [#UnitFB];

NETWORK
TITLE =A9_UV1  Bypass CIP Anlage 9
// Act 019
// Box           : VSRVK1..3
// Input address : I82.4
// Output address: Q82.4
      CALL FC    70 (
           UnitNo                   := #UnitNo,
           ActRec                   := DB2690.A9_UV1,
           Typ                      := 1,
           FBa                      := #xTmp,
           FBa2                     := I     82.4,
           Out                      := Q     82.4);

NETWORK
TITLE =A9_RR1  Reinigungsrücklauf Anlage 9 zu Kreis 1
// Act 020
// Box           : VSRR1-3
// Input address : I84.3
// Output address: Q84.3
      CALL FC    70 (
           UnitNo                   := #UnitNo,
           ActRec                   := DB2690.A9_RR1,
           Typ                      := 1,
           FBa                      := #xTmp,
           FBa2                     := I     84.3,
           Out                      := Q     84.3);

NETWORK
TITLE =A9_RR2  Reinigungsrücklauf Anlage 9 zu Kreis 2
// Act 021
// Box           : VSRR1-3
// Input address : I84.4
// Output address: Q84.4
      CALL FC    70 (
           UnitNo                   := #UnitNo,
           ActRec                   := DB2690.A9_RR2,
           Typ                      := 1,
           FBa                      := #xTmp,
           FBa2                     := I     84.4,
           Out                      := Q     84.4);

NETWORK
TITLE =A9_RR3  Reinigungsrücklauf Anlage 9 zu Kreis 3
// Act 022
// Box           : VSRR1-3
// Input address : I84.5
// Output address: Q84.5
      CALL FC    70 (
           UnitNo                   := #UnitNo,
           ActRec                   := DB2690.A9_RR3,
           Typ                      := 1,
           FBa                      := #xTmp,
           FBa2                     := I     84.5,
           Out                      := Q     84.5);

NETWORK
TITLE =LA_LDS_A9_V11  AB FUELLER 9/10
// Act 023
// Box           : S8 U8.2
// Input address : I52.0
// Output address: Q111.5
      CALL FC    70 (
           UnitNo                   := #UnitNo,
           ActRec                   := DB2690.LA_LDS_A9_V11,
           Typ                      := 0,
           FBa                      := #xTmp,
           FBa2                     := I     52.0,
           Out                      := Q    111.5);

NETWORK
TITLE =LA_LDS_A9_V12  AB FUELLER 9/10
// Act 024
// Box           : S8 U8.2
// Input address : I52.1
// Output address: Q111.6
      CALL FC    70 (
           UnitNo                   := #UnitNo,
           ActRec                   := DB2690.LA_LDS_A9_V12,
           Typ                      := 0,
           FBa                      := #xTmp,
           FBa2                     := I     52.1,
           Out                      := Q    111.6);

NETWORK
TITLE =LA_LDS_A9_V13  AB FUELLER 9/10
// Act 025
// Box           : S8 U8.2
// Input address : I52.2
// Output address: Q111.7
      CALL FC    70 (
           UnitNo                   := #UnitNo,
           ActRec                   := DB2690.LA_LDS_A9_V13,
           Typ                      := 0,
           FBa                      := #xTmp,
           FBa2                     := I     52.2,
           Out                      := Q    111.7);

NETWORK
TITLE =RUECKL_ROEHRE_SPUELF9  SIGNAL AN FUELLER 9
// Act 026
// Box           : S8 U8.2
// Output address: Q40.6
      CALL FC    70 (
           UnitNo                   := #UnitNo,
           ActRec                   := DB2690.RUECKL_ROEHRE_SPUELF9,
           Typ                      := 0,
           FBa                      := #xTmp,
           FBa2                     := #xTmp,
           Out                      := Q     40.6);

NETWORK
TITLE =RUECKL_ROEHRE_SPUELF10  SIGNAL AN FUELLER 10
// Act 027
// Box           : S8 U8.2
// Output address: Q40.7
      CALL FC    70 (
           UnitNo                   := #UnitNo,
           ActRec                   := DB2690.RUECKL_ROEHRE_SPUELF10,
           Typ                      := 0,
           FBa                      := #xTmp,
           FBa2                     := #xTmp,
           Out                      := Q     40.7);

NETWORK
TITLE =UMSCHALTSIGN_MIX_F9_10  SIGNAL AN MIXER F9/10
// Act 029
// Box           : S8 U8.2
// Output address: Q41.2
      CALL FC    70 (
           UnitNo                   := #UnitNo,
           ActRec                   := DB2690.UMSCHALTSIGN_MIX_F9_10,
           Typ                      := 0,
           FBa                      := #xTmp,
           FBa2                     := #xTmp,
           Out                      := Q     41.2);

NETWORK
TITLE =STOP_SIGNALMIX_F9_10  SIGNAL AN MIXER F9/10
// Act 030
// Box           : S8 U8.2
// Output address: Q41.3
      CALL FC    70 (
           UnitNo                   := #UnitNo,
           ActRec                   := DB2690.STOP_SIGNALMIX_F9_10,
           Typ                      := 0,
           FBa                      := #xTmp,
           FBa2                     := #xTmp,
           Out                      := Q     41.3);

NETWORK
TITLE =HF9V2_OFFEN_MIX_F9_10  SIGNAL AN MIXER F9/10
// Act 031
// Box           : S8 U8.2
// Output address: Q41.4
      CALL FC    70 (
           UnitNo                   := #UnitNo,
           ActRec                   := DB2690.HF9V2_OFFEN_MIX_F9_10,
           Typ                      := 0,
           FBa                      := #xTmp,
           FBa2                     := #xTmp,
           Out                      := Q     41.4);

NETWORK
TITLE =LA_LDT_A9_CIP  AB FUELLER 9/10
// Act 035
// Box           : S8 U8.2
// Output address: Q42.6
      CALL FC    70 (
           UnitNo                   := #UnitNo,
           ActRec                   := DB2690.LA_LDT_A9_CIP,
           Typ                      := 0,
           FBa                      := #xTmp,
           FBa2                     := #xTmp,
           Out                      := Q     42.6);

NETWORK
TITLE =LA_A9_TSH  AB FUELLER 9/10
// Act 036
// Box           : S8 U8.2
// Output address: Q42.7
      CALL FC    70 (
           UnitNo                   := #UnitNo,
           ActRec                   := DB2690.LA_A9_TSH,
           Typ                      := 0,
           FBa                      := #xTmp,
           FBa2                     := #xTmp,
           Out                      := Q     42.7);

NETWORK
TITLE =HEISSABFUELUNG_OK_F9  SIGNAL VON TU AN FUELLER 9
// Act 037
// Box           : S8 U8.2
// Output address: Q43.6
      CALL FC    70 (
           UnitNo                   := #UnitNo,
           ActRec                   := DB2690.HEISSABFUELUNG_OK_F9,
           Typ                      := 0,
           FBa                      := #xTmp,
           FBa2                     := #xTmp,
           Out                      := Q     43.6);

NETWORK
TITLE =LA_LDT_A9PRODUKT  AB FUELLER 9/10
// Act 038
// Box           : S8 U8.2
// Output address: Q43.7
      CALL FC    70 (
           UnitNo                   := #UnitNo,
           ActRec                   := DB2690.LA_LDT_A9PRODUKT,
           Typ                      := 0,
           FBa                      := #xTmp,
           FBa2                     := #xTmp,
           Out                      := Q     43.7);

NETWORK
TITLE =F9_LEERDRUECKEN  SIGNAL VON TU AN FUELLER 9
// Act 039
// Box           : S8 U8.2
// Output address: Q120.0
      CALL FC    70 (
           UnitNo                   := #UnitNo,
           ActRec                   := DB2690.F9_LEERDRUECKEN,
           Typ                      := 0,
           FBa                      := #xTmp,
           FBa2                     := #xTmp,
           Out                      := Q    120.0);

NETWORK
TITLE =F9_AUF_KREISLAUF  SIGNAL VON TU AN FUELLER 9
// Act 040
// Box           : S8 U8.2
// Output address: Q120.1
      CALL FC    70 (
           UnitNo                   := #UnitNo,
           ActRec                   := DB2690.F9_AUF_KREISLAUF,
           Typ                      := 0,
           FBa                      := #xTmp,
           FBa2                     := #xTmp,
           Out                      := Q    120.1);

END_FUNCTION_BLOCK

FUNCTION_BLOCK FB 1691
TITLE =U069: Packaging Plant 9
FAMILY : BOTEC_F1
NAME : UniE
VERSION : 1.2


VAR_TEMP
  CIP : BOOL ;	//CIP active
  UNIM : BOOL ;	//Unit Not In Maintenance
  GenRel : BOOL ;	//general OK (emergency and maintenance OK)
  EStopOK : BOOL ;	//emergency OK
  UnitNo : INT ;	//unit number
  xTmp : BOOL ;	//Temporary Bool
  iTmp : INT ;	//Temporary INT
  rTmp : REAL ;	//Temporary REAL
  dTmp : DINT ;	//Temporary DINT (free for general use)
  RetValInt : INT ;	//return value
END_VAR
BEGIN
NETWORK
TITLE =General

      SET   ;
// Simulation ---------------------------------------------------------------
      A     DB1691.DBX 1357.7;
      CC    FB  1699; // "U069Sim"
      A     DB1691.DBX   17.3;
      =     DB1691.DBX 1357.7; //Help bit for simulation

// get unit number ----------------------------------------------------------
      L     DB1690.DBW    0;
      T     #UnitNo;

// CIP ----------------------------------------------------------------------
      L     DB1691.DBD   54;
      L     0;
      <D    ;
      =     #CIP;

// emergency OK -------------------------------------------------------------
      A     DB1695.DBX   27.0; //Emergency Stop OK
      =     #EStopOK;

// Write Unit in Maintenance ------------------------------------------------

      AN    DB1691.DBX   69.7;
      =     #UNIM;

// emergency and maintenance OK ---------------------------------------------
      A     #EStopOK;
      A     #UNIM;
      =     #GenRel;

// communication ------------------------------------------------------------
      UC    FB  1695; // U069Com

NETWORK
TITLE =Analog Inputs

      NOP   0;

// ----------------------------------------------------------
// HWWT1_TT01 Heißwasser-Wärmetauscher1 TT01
// ----------------------------------------------------------
      L     DB1691.DBD 1118; // !!! insert correct SFM !!!
      T     DB2693.DBD  238;

//      SET
//      =     "U069AnID".HWWT1_TT01.EAlHH

NETWORK
TITLE =Universal Value

      NOP   0;

// ----------------------------------------------------------
// unv001 Process Status
// ----------------------------------------------------------
// process value to UnV
//      L     0.000000e+000
//      T     "U069UnVD".unv001.ValExt

// ----------------------------------------------------------
// unv002 Universal Value 02
// ----------------------------------------------------------
// process value to UnV
//      L     0.000000e+000
//      T     "U069UnVD".unv002.ValExt

// ----------------------------------------------------------
// unv003 Universal Value 03
// ----------------------------------------------------------
// process value to UnV
//      L     0.000000e+000
//      T     "U069UnVD".unv003.ValExt

// ----------------------------------------------------------
// unv004 Universal Value 04
// ----------------------------------------------------------
// process value to UnV
//      L     0.000000e+000
//      T     "U069UnVD".unv004.ValExt

NETWORK
TITLE =Special Input

      NOP   0;

// ----------------------------------------------------------
// LS_LLL_A9 SIGNAL VON FUELLER 9
// ----------------------------------------------------------
//      CLR
//      =     "U069SpID".LS_LLL_A9.EAl
//      =     "U069SpID".LS_LLL_A9.Pre

// ----------------------------------------------------------
// TS_HL_ANL9
// ----------------------------------------------------------
//      CLR
//      =     "U069SpID".TS_HL_ANL9.EAl
//      =     "U069SpID".TS_HL_ANL9.Pre

// ----------------------------------------------------------
// A9_SS_FRG_MOLCH Anlage 9 Schlüsselschalter Freigabe Molch
// ----------------------------------------------------------
//      CLR
//      =     "U069SpID".A9_SS_FRG_MOLCH.EAl
//      =     "U069SpID".A9_SS_FRG_MOLCH.Pre

// ----------------------------------------------------------
// LDT_A9_PRODUKT AB FUELLER 9/10
// ----------------------------------------------------------
//      CLR
//      =     "U069SpID".LDT_A9_PRODUKT.EAl
//      =     "U069SpID".LDT_A9_PRODUKT.Pre

// ----------------------------------------------------------
// LDT_A9_CIP AB FUELLER 9/10
// ----------------------------------------------------------
//      CLR
//      =     "U069SpID".LDT_A9_CIP.EAl
//      =     "U069SpID".LDT_A9_CIP.Pre

// ----------------------------------------------------------
// DT_A9_START AB FUELLER 9/10
// ----------------------------------------------------------
//      CLR
//      =     "U069SpID".DT_A9_START.EAl
//      =     "U069SpID".DT_A9_START.Pre

// ----------------------------------------------------------
// DT_A9_STOP AB FUELLER 9/10
// ----------------------------------------------------------
//      CLR
//      =     "U069SpID".DT_A9_STOP.EAl
//      =     "U069SpID".DT_A9_STOP.Pre

// ----------------------------------------------------------
// DT_LAMPEN_PRUEFEN_A9_L10 AB FUELLER 9/10
// ----------------------------------------------------------
//      CLR
//      =     "U069SpID".DT_LAMPEN_PRUEFEN_A9_L10.EAl
//      =     "U069SpID".DT_LAMPEN_PRUEFEN_A9_L10.Pre

// ----------------------------------------------------------
// QUITT_A9_LA10
// ----------------------------------------------------------
//      CLR
//      =     "U069SpID".QUITT_A9_LA10.EAl
//      =     "U069SpID".QUITT_A9_LA10.Pre

// ----------------------------------------------------------
// BETRIEB_F9 SIGNAL VON FUELLER 9
// ----------------------------------------------------------
//      CLR
//      =     "U069SpID".BETRIEB_F9.EAl
//      =     "U069SpID".BETRIEB_F9.Pre

// ----------------------------------------------------------
// BETRIEB_MIX_LKASKADE_F9 SIGNAL VON FUELLER 9
// ----------------------------------------------------------
//      CLR
//      =     "U069SpID".BETRIEB_MIX_LKASKADE_F9.EAl
//      =     "U069SpID".BETRIEB_MIX_LKASKADE_F9.Pre

// ----------------------------------------------------------
// M9_Produkt_kommt Meldung von Mixer9 für Heißabfüllung-Ausschub
// ----------------------------------------------------------
//      CLR
//      =     "U069SpID".M9_Produkt_kommt.EAl
//      =     "U069SpID".M9_Produkt_kommt.Pre

// ----------------------------------------------------------
// F9_TEMPERATUR_ERREICHT SIGNAL VON FUELLER 9
// ----------------------------------------------------------
//      CLR
//      =     "U069SpID".F9_TEMPERATUR_ERREICHT.EAl
//      =     "U069SpID".F9_TEMPERATUR_ERREICHT.Pre

// ----------------------------------------------------------
// F9_TEMPERATUR_MIN_LMAX SIGNAL VON FUELLER 9
// ----------------------------------------------------------
//      CLR
//      =     "U069SpID".F9_TEMPERATUR_MIN_LMAX.EAl
//      =     "U069SpID".F9_TEMPERATUR_MIN_LMAX.Pre

// ----------------------------------------------------------
// F9_ANF_PRODUKTPUMPE SIGNAL VON FUELLER 9
// ----------------------------------------------------------
//      CLR
//      =     "U069SpID".F9_ANF_PRODUKTPUMPE.EAl
//      =     "U069SpID".F9_ANF_PRODUKTPUMPE.Pre

// ----------------------------------------------------------
// F9_PRODUKTIONSENDE SIGNAL VON FUELLER 9
// ----------------------------------------------------------
//      CLR
//      =     "U069SpID".F9_PRODUKTIONSENDE.EAl
//      =     "U069SpID".F9_PRODUKTIONSENDE.Pre

// ----------------------------------------------------------
// F9_BETRIEBSBEREIT SIGNAL VON FUELLER 9
// ----------------------------------------------------------
//      CLR
//      =     "U069SpID".F9_BETRIEBSBEREIT.EAl
//      =     "U069SpID".F9_BETRIEBSBEREIT.Pre

// ----------------------------------------------------------
// RM_RWPA9 SIGNAL VON MIXER F9/10
// ----------------------------------------------------------
//      CLR
//      =     "U069SpID".RM_RWPA9.EAl
//      =     "U069SpID".RM_RWPA9.Pre

// ----------------------------------------------------------
// MIX_WEGFREIGABE_9_L9 SIGNAL VON MIXER A9/10
// ----------------------------------------------------------
//      CLR
//      =     "U069SpID".MIX_WEGFREIGABE_9_L9.EAl
//      =     "U069SpID".MIX_WEGFREIGABE_9_L9.Pre

// ----------------------------------------------------------
// MIX_WEGFREIGABE_9_L10 SIGNAL VON MIXER A9/10
// ----------------------------------------------------------
//      CLR
//      =     "U069SpID".MIX_WEGFREIGABE_9_L10.EAl
//      =     "U069SpID".MIX_WEGFREIGABE_9_L10.Pre

// ----------------------------------------------------------
// MIX_ANFORDERUNG_PUMPE SIGNAL VON MIXER F9/F10
// ----------------------------------------------------------
//      CLR
//      =     "U069SpID".MIX_ANFORDERUNG_PUMPE.EAl
//      =     "U069SpID".MIX_ANFORDERUNG_PUMPE.Pre

NETWORK
TITLE =Messages

      NOP   0;

// ----------------------------------------------------------
// msg001 Message 01
// ----------------------------------------------------------
      SET   ;
      R     DB2697.DBX   80.7;
      =     DB2697.DBX   81.4;

      CLR   ;
      =     DB2697.DBX   82.7;

